LIN {X 0,Y 354.797,Z 576.907,A -85,B 0,C 180,E1 -13637.677,E2 -13637.677} C_VEL
LIN {X 0,Y 353.778,Z 635.743,A -85,B 0,C 180,E1 -13639.096,E2 -13639.096} C_VEL
LIN {X 0,Y 353.628,Z 649.216,A -85,B 0,C 180,E1 -13639.603,E2 -13639.603} C_VEL
LIN {X 0,Y 353.219,Z 662.716,A -85,B 0,C 180,E1 -13640.361,E2 -13640.361} C_VEL
LIN {X 0,Y 352.689,Z 674.449,A -85,B 0,C 180,E1 -13641.241,E2 -13641.241} C_VEL
LIN {X 0,Y 352.081,Z 686.1,A -85,B 0,C 180,E1 -13642.369,E2 -13642.369} C_VEL
LIN {X 0,Y 351.35,Z 696.823,A -85,B 0,C 180,E1 -13643.659,E2 -13643.659} C_VEL
LIN {X 0,Y 350.663,Z 705.588,A -85,B 0,C 180,E1 -13644.945,E2 -13644.945} C_VEL
LIN {X 0,Y 349.989,Z 714.199,A -85,B 0,C 180,E1 -13646.481,E2 -13646.481} C_VEL
LIN {X 0,Y 349.423,Z 721.312,A -85,B 0,C 180,E1 -13648.03,E2 -13648.03} C_VEL
LIN {X 0,Y 348.756,Z 728.774,A -85,B 0,C 180,E1 -13650.053,E2 -13650.053} C_VEL
LIN {X 0,Y 348.488,Z 733.524,A -85,B 0,C 180,E1 -13651.71,E2 -13651.71} C_VEL
LIN {X 0,Y 348.166,Z 737.758,A -85,B 0,C 180,E1 -13653.635,E2 -13653.635} C_VEL
LIN {X 0,Y 348.044,Z 740.417,A -85,B 0,C 180,E1 -13655.319,E2 -13655.319} C_VEL
LIN {X 0,Y 348.012,Z 742.443,A -85,B 0,C 180,E1 -13657.437,E2 -13657.437} C_VEL
LIN {X 0,Y 348.114,Z 743.004,A -85,B 0,C 180,E1 -13658.691,E2 -13658.691} C_VEL
LIN {X 0,Y 348.273,Z 743.074,A -85,B 0,C 180,E1 -13659.937,E2 -13659.937} C_VEL
LIN {X 0,Y 348.516,Z 742.538,A -85,B 0,C 180,E1 -13661.396,E2 -13661.396} C_VEL
LIN {X 0,Y 348.724,Z 741.797,A -85,B 0,C 180,E1 -13662.404,E2 -13662.404} C_VEL
LIN {X 0,Y 349.092,Z 740.415,A -85,B 0,C 180,E1 -13663.629,E2 -13663.629} C_VEL
LIN {X 0,Y 349.712,Z 737.457,A -85,B 0,C 180,E1 -13665.451,E2 -13665.451} C_VEL
LIN {X 0,Y 350.505,Z 733.331,A -85,B 0,C 180,E1 -13667.258,E2 -13667.258} C_VEL
LIN {X 0,Y 351.534,Z 727.601,A -85,B 0,C 180,E1 -13669.148,E2 -13669.148} C_VEL
LIN {X 0,Y 352.555,Z 721.084,A -85,B 0,C 180,E1 -13670.823,E2 -13670.823} C_VEL
LIN {X 0,Y 353.791,Z 712.466,A -85,B 0,C 180,E1 -13672.582,E2 -13672.582} C_VEL
LIN {X 0,Y 354.949,Z 703.421,A -85,B 0,C 180,E1 -13674.064,E2 -13674.064} C_VEL
LIN {X 0,Y 356.03,Z 693.807,A -85,B 0,C 180,E1 -13675.329,E2 -13675.329} C_VEL
LIN {X 0,Y 357.056,Z 682.997,A -85,B 0,C 180,E1 -13676.473,E2 -13676.473} C_VEL
LIN {X 0,Y 357.886,Z 671.118,A -85,B 0,C 180,E1 -13677.468,E2 -13677.468} C_VEL
LIN {X 0,Y 358.466,Z 657.986,A -85,B 0,C 180,E1 -13678.284,E2 -13678.284} C_VEL
LIN {X 0,Y 358.763,Z 645.264,A -85,B 0,C 180,E1 -13678.843,E2 -13678.843} C_VEL
LIN {X 0,Y 359.132,Z 620.722,A -85,B 0,C 180,E1 -13679.534,E2 -13679.534} C_VEL
LIN {X 0,Y 360.495,Z 582.186,A -85,B 0,C 180,E1 -13680.545,E2 -13680.545} C_VEL
LIN {X 0,Y 354.117,Z 568.659,A -85,B 0,C 180,E1 -13681.601,E2 -13681.601} C_VEL
LIN {X 0,Y 349.417,Z 560.316,A -85,B 0,C 180,E1 -13682.383,E2 -13682.383} C_VEL
LIN {X 0,Y 348.227,Z 557.698,A -85,B 0,C 180,E1 -13682.603,E2 -13682.603} C_VEL
LIN {X 0,Y 348.11,Z 557.127,A -85,B 0,C 180,E1 -13682.676,E2 -13682.676} C_VEL
LIN {X 0,Y 348.099,Z 557.121,A -85,B 0,C 180,E1 -13686.958,E2 -13686.958} C_VEL
LIN {X 0,Y 347.959,Z 557.14,A -85,B 0,C 180,E1 -13689.299,E2 -13689.299} C_VEL
LIN {X 0,Y 347.884,Z 557.146,A -85,B 0,C 180,E1 -13692.84,E2 -13692.84} C_VEL
LIN {X 0,Y 347.829,Z 557.152,A -85,B 0,C 180,E1 -13696.432,E2 -13696.432} C_VEL
LIN {X 0,Y 347.846,Z 557.158,A -85,B 0,C 180,E1 -13698.861,E2 -13698.861} C_VEL
LIN {X 0,Y 347.765,Z 557.166,A -85,B 0,C 180,E1 -13702.58,E2 -13702.58} C_VEL
LIN {X 0,Y 347.803,Z 557.162,A -85,B 0,C 180,E1 -13705.109,E2 -13705.109} C_VEL
LIN {X 0,Y 347.803,Z 557.158,A -85,B 0,C 180,E1 -13707.695,E2 -13707.695} C_VEL
LIN {X 0,Y 347.756,Z 557.168,A -85,B 0,C 180,E1 -13710.347,E2 -13710.347} C_VEL
LIN {X 0,Y 347.736,Z 557.164,A -85,B 0,C 180,E1 -13714.465,E2 -13714.465} C_VEL
LIN {X 0,Y 347.769,Z 557.161,A -85,B 0,C 180,E1 -13717.99,E2 -13717.99} C_VEL
LIN {X 0,Y 347.778,Z 557.167,A -85,B 0,C 180,E1 -13721.61,E2 -13721.61} C_VEL
LIN {X 0,Y 347.825,Z 557.158,A -85,B 0,C 180,E1 -13725.007,E2 -13725.007} C_VEL
LIN {X 0,Y 347.779,Z 557.165,A -85,B 0,C 180,E1 -13728.392,E2 -13728.392} C_VEL
LIN {X 0,Y 347.801,Z 557.245,A -85,B 0,C 180,E1 -13731.216,E2 -13731.216} C_VEL
LIN {X 0,Y 351.006,Z 568.194,A -85,B 0,C 180,E1 -13734.506,E2 -13734.506} C_VEL
LIN {X 0,Y 353.622,Z 578.805,A -85,B 0,C 180,E1 -13737.302,E2 -13737.302} C_VEL
LIN {X 0,Y 355.347,Z 587.427,A -85,B 0,C 180,E1 -13739.386,E2 -13739.386} C_VEL
LIN {X 0,Y 355.219,Z 590.506,A -85,B 0,C 180,E1 -13740.03,E2 -13740.03} C_VEL
LIN {X 0,Y 352.496,Z 610.75,A -85,B 0,C 180,E1 -13743.985,E2 -13743.985} C_VEL
LIN {X 0,Y 351.698,Z 617.716,A -85,B 0,C 180,E1 -13745.318,E2 -13745.318} C_VEL
LIN {X 0,Y 355.284,Z 641.232,A -85,B 0,C 180,E1 -13746.39,E2 -13746.39} C_VEL
LIN {X 0,Y 357.422,Z 662.797,A -85,B 0,C 180,E1 -13747.201,E2 -13747.201} C_VEL
LIN {X 0,Y 358.192,Z 678.894,A -85,B 0,C 180,E1 -13747.723,E2 -13747.723} C_VEL
LIN {X 0,Y 356.353,Z 732.757,A -85,B 0,C 180,E1 -13749.097,E2 -13749.097} C_VEL
LIN {X 0,Y 355.4,Z 746.792,A -85,B 0,C 180,E1 -13749.679,E2 -13749.679} C_VEL
LIN {X 0,Y 355.085,Z 750.828,A -85,B 0,C 180,E1 -13749.849,E2 -13749.849} C_VEL
LIN {X 0,Y 354.525,Z 764.15,A -85,B 0,C 180,E1 -13750.269,E2 -13750.269} C_VEL
LIN {X 0,Y 353.732,Z 776.246,A -85,B 0,C 180,E1 -13750.865,E2 -13750.865} C_VEL
LIN {X 0,Y 352.774,Z 788.474,A -85,B 0,C 180,E1 -13751.715,E2 -13751.715} C_VEL
LIN {X 0,Y 351.717,Z 799.465,A -85,B 0,C 180,E1 -13752.71,E2 -13752.71} C_VEL
LIN {X 0,Y 350.555,Z 810.407,A -85,B 0,C 180,E1 -13753.965,E2 -13753.965} C_VEL
LIN {X 0,Y 349.407,Z 820.549,A -85,B 0,C 180,E1 -13755.439,E2 -13755.439} C_VEL
LIN {X 0,Y 348.514,Z 828.654,A -85,B 0,C 180,E1 -13756.889,E2 -13756.889} C_VEL
LIN {X 0,Y 347.567,Z 836.584,A -85,B 0,C 180,E1 -13758.631,E2 -13758.631} C_VEL
LIN {X 0,Y 347.055,Z 841.938,A -85,B 0,C 180,E1 -13760.09,E2 -13760.09} C_VEL
LIN {X 0,Y 346.613,Z 847.165,A -85,B 0,C 180,E1 -13761.841,E2 -13761.841} C_VEL
LIN {X 0,Y 346.333,Z 851.786,A -85,B 0,C 180,E1 -13763.902,E2 -13763.902} C_VEL
LIN {X 0,Y 346.288,Z 854.185,A -85,B 0,C 180,E1 -13765.345,E2 -13765.345} C_VEL
LIN {X 0,Y 346.225,Z 855.612,A -85,B 0,C 180,E1 -13766.51,E2 -13766.51} C_VEL
LIN {X 0,Y 346.248,Z 857.236,A -85,B 0,C 180,E1 -13768.838,E2 -13768.838} C_VEL
LIN {X 0,Y 346.311,Z 857.456,A -85,B 0,C 180,E1 -13770.001,E2 -13770.001} C_VEL
LIN {X 0,Y 346.228,Z 857.23,A -85,B 0,C 180,E1 -13771.164,E2 -13771.164} C_VEL
LIN {X 0,Y 346.216,Z 855.598,A -85,B 0,C 180,E1 -13773.492,E2 -13773.492} C_VEL
LIN {X 0,Y 346.279,Z 854.163,A -85,B 0,C 180,E1 -13774.657,E2 -13774.657} C_VEL
LIN {X 0,Y 346.307,Z 851.838,A -85,B 0,C 180,E1 -13776.058,E2 -13776.058} C_VEL
LIN {X 0,Y 346.61,Z 847.128,A -85,B 0,C 180,E1 -13778.161,E2 -13778.161} C_VEL
LIN {X 0,Y 347.137,Z 840.879,A -85,B 0,C 180,E1 -13780.205,E2 -13780.205} C_VEL
LIN {X 0,Y 347.798,Z 834.061,A -85,B 0,C 180,E1 -13781.955,E2 -13781.955} C_VEL
LIN {X 0,Y 348.86,Z 825.532,A -85,B 0,C 180,E1 -13783.693,E2 -13783.693} C_VEL
LIN {X 0,Y 349.858,Z 816.746,A -85,B 0,C 180,E1 -13785.139,E2 -13785.139} C_VEL
LIN {X 0,Y 350.833,Z 807.081,A -85,B 0,C 180,E1 -13786.437,E2 -13786.437} C_VEL
LIN {X 0,Y 351.991,Z 796.48,A -85,B 0,C 180,E1 -13787.578,E2 -13787.578} C_VEL
LIN {X 0,Y 353.108,Z 784.571,A -85,B 0,C 180,E1 -13788.57,E2 -13788.57} C_VEL
LIN {X 0,Y 353.992,Z 772.163,A -85,B 0,C 180,E1 -13789.349,E2 -13789.349} C_VEL
LIN {X 0,Y 354.749,Z 760.169,A -85,B 0,C 180,E1 -13789.871,E2 -13789.871} C_VEL
LIN {X 0,Y 355.231,Z 746.868,A -85,B 0,C 180,E1 -13790.22,E2 -13790.22} C_VEL
LIN {X 0,Y 356.311,Z 677.092,A -85,B 0,C 180,E1 -13791.622,E2 -13791.622} C_VEL
LIN {X 0,Y 352.473,Z 643.046,A -85,B 0,C 180,E1 -13792.599,E2 -13792.599} C_VEL
LIN {X 0,Y 351.528,Z 636.097,A -85,B 0,C 180,E1 -13792.83,E2 -13792.83} C_VEL
LIN {X 0,Y 350.218,Z 619.795,A -85,B 0,C 180,E1 -13793.899,E2 -13793.899} C_VEL
LIN {X 0,Y 352.061,Z 599.692,A -85,B 0,C 180,E1 -13797.978,E2 -13797.978} C_VEL
LIN {X 0,Y 353.609,Z 584.378,A -85,B 0,C 180,E1 -13801.115,E2 -13801.115} C_VEL
LIN {X 0,Y 351.574,Z 574.031,A -85,B 0,C 180,E1 -13803.456,E2 -13803.456} C_VEL
LIN {X 0,Y 348.306,Z 559.575,A -85,B 0,C 180,E1 -13806.864,E2 -13806.864} C_VEL
LIN {X 0,Y 347.787,Z 557.165,A -85,B 0,C 180,E1 -13807.485,E2 -13807.485} C_VEL
LIN {X 0,Y 347.735,Z 557.17,A -85,B 0,C 180,E1 -13810.297,E2 -13810.297} C_VEL
LIN {X 0,Y 347.725,Z 557.162,A -85,B 0,C 180,E1 -13813.408,E2 -13813.408} C_VEL
LIN {X 0,Y 347.73,Z 557.171,A -85,B 0,C 180,E1 -13816.686,E2 -13816.686} C_VEL
LIN {X 0,Y 347.749,Z 557.166,A -85,B 0,C 180,E1 -13820.173,E2 -13820.173} C_VEL
LIN {X 0,Y 347.764,Z 557.157,A -85,B 0,C 180,E1 -13822.679,E2 -13822.679} C_VEL
LIN {X 0,Y 347.75,Z 557.167,A -85,B 0,C 180,E1 -13825.956,E2 -13825.956} C_VEL
LIN {X 0,Y 347.765,Z 557.153,A -85,B 0,C 180,E1 -13829.654,E2 -13829.654} C_VEL
LIN {X 0,Y 347.853,Z 557.154,A -85,B 0,C 180,E1 -13832.745,E2 -13832.745} C_VEL
LIN {X 0,Y 347.787,Z 557.151,A -85,B 0,C 180,E1 -13836.162,E2 -13836.162} C_VEL
LIN {X 0,Y 347.808,Z 557.155,A -85,B 0,C 180,E1 -13839.909,E2 -13839.909} C_VEL
LIN {X 0,Y 347.867,Z 557.131,A -85,B 0,C 180,E1 -13842.359,E2 -13842.359} C_VEL
LIN {X 0,Y 347.899,Z 557.148,A -85,B 0,C 180,E1 -13845.971,E2 -13845.971} C_VEL
LIN {X 0,Y 347.929,Z 557.124,A -85,B 0,C 180,E1 -13849.526,E2 -13849.526} C_VEL
LIN {X 0,Y 348.093,Z 557.123,A -85,B 0,C 180,E1 -13853.042,E2 -13853.042} C_VEL
LIN {X 0,Y 348.206,Z 557.089,A -85,B 0,C 180,E1 -13857.687,E2 -13857.687} C_VEL
LIN {X 0,Y 348.325,Z 557.095,A -85,B 0,C 180,E1 -13860,E2 -13860} C_VEL
LIN {X 0,Y 348.207,Z 557.106,A -85,B 0,C 180,E1 -13862.314,E2 -13862.314} C_VEL
LIN {X 0,Y 348.094,Z 557.116,A -85,B 0,C 180,E1 -13866.958,E2 -13866.958} C_VEL
LIN {X 0,Y 347.931,Z 557.137,A -85,B 0,C 180,E1 -13870.474,E2 -13870.474} C_VEL
LIN {X 0,Y 347.9,Z 557.141,A -85,B 0,C 180,E1 -13874.15,E2 -13874.15} C_VEL
LIN {X 0,Y 347.892,Z 557.135,A -85,B 0,C 180,E1 -13878.29,E2 -13878.29} C_VEL
LIN {X 0,Y 347.79,Z 557.16,A -85,B 0,C 180,E1 -13881.635,E2 -13881.635} C_VEL
LIN {X 0,Y 347.813,Z 557.145,A -85,B 0,C 180,E1 -13885.108,E2 -13885.108} C_VEL
LIN {X 0,Y 347.81,Z 557.159,A -85,B 0,C 180,E1 -13887.694,E2 -13887.694} C_VEL
LIN {X 0,Y 347.751,Z 557.156,A -85,B 0,C 180,E1 -13890.348,E2 -13890.348} C_VEL
LIN {X 0,Y 347.75,Z 557.168,A -85,B 0,C 180,E1 -13894.044,E2 -13894.044} C_VEL
LIN {X 0,Y 347.763,Z 557.167,A -85,B 0,C 180,E1 -13897.321,E2 -13897.321} C_VEL
LIN {X 0,Y 347.734,Z 557.167,A -85,B 0,C 180,E1 -13900.297,E2 -13900.297} C_VEL
LIN {X 0,Y 347.725,Z 557.163,A -85,B 0,C 180,E1 -13903.408,E2 -13903.408} C_VEL
LIN {X 0,Y 347.727,Z 557.152,A -85,B 0,C 180,E1 -13906.686,E2 -13906.686} C_VEL
LIN {X 0,Y 347.751,Z 557.17,A -85,B 0,C 180,E1 -13910.173,E2 -13910.173} C_VEL
LIN {X 0,Y 347.765,Z 557.155,A -85,B 0,C 180,E1 -13912.679,E2 -13912.679} C_VEL
LIN {X 0,Y 347.804,Z 557.278,A -85,B 0,C 180,E1 -13915.058,E2 -13915.058} C_VEL
LIN {X 0,Y 351.695,Z 571.483,A -85,B 0,C 180,E1 -13918.025,E2 -13918.025} C_VEL
LIN {X 0,Y 354.731,Z 584.606,A -85,B 0,C 180,E1 -13920.662,E2 -13920.662} C_VEL
LIN {X 0,Y 355.49,Z 588.601,A -85,B 0,C 180,E1 -13921.437,E2 -13921.437} C_VEL
LIN {X 0,Y 354.195,Z 606.433,A -85,B 0,C 180,E1 -13924.432,E2 -13924.432} C_VEL
LIN {X 0,Y 353.21,Z 623.88,A -85,B 0,C 180,E1 -13927.211,E2 -13927.211} C_VEL
LIN {X 0,Y 357.261,Z 649.9,A -85,B 0,C 180,E1 -13928.051,E2 -13928.051} C_VEL
LIN {X 0,Y 355.98,Z 721.054,A -85,B 0,C 180,E1 -13929.486,E2 -13929.486} C_VEL
LIN {X 0,Y 355.648,Z 737.977,A -85,B 0,C 180,E1 -13929.881,E2 -13929.881} C_VEL
LIN {X 0,Y 354.963,Z 751.645,A -85,B 0,C 180,E1 -13930.443,E2 -13930.443} C_VEL
LIN {X 0,Y 354.078,Z 763.979,A -85,B 0,C 180,E1 -13931.183,E2 -13931.183} C_VEL
LIN {X 0,Y 353.008,Z 776.117,A -85,B 0,C 180,E1 -13932.175,E2 -13932.175} C_VEL
LIN {X 0,Y 351.907,Z 787.509,A -85,B 0,C 180,E1 -13933.377,E2 -13933.377} C_VEL
LIN {X 0,Y 350.973,Z 796.862,A -85,B 0,C 180,E1 -13934.615,E2 -13934.615} C_VEL
LIN {X 0,Y 349.814,Z 805.738,A -85,B 0,C 180,E1 -13936.048,E2 -13936.048} C_VEL
LIN {X 0,Y 348.749,Z 814.393,A -85,B 0,C 180,E1 -13937.783,E2 -13937.783} C_VEL
LIN {X 0,Y 347.875,Z 821.352,A -85,B 0,C 180,E1 -13939.523,E2 -13939.523} C_VEL
LIN {X 0,Y 347.175,Z 826.884,A -85,B 0,C 180,E1 -13941.266,E2 -13941.266} C_VEL
LIN {X 0,Y 346.719,Z 831.878,A -85,B 0,C 180,E1 -13943.333,E2 -13943.333} C_VEL
LIN {X 0,Y 346.422,Z 835.356,A -85,B 0,C 180,E1 -13945.344,E2 -13945.344} C_VEL
LIN {X 0,Y 346.254,Z 836.779,A -85,B 0,C 180,E1 -13946.508,E2 -13946.508} C_VEL
LIN {X 0,Y 346.155,Z 838.388,A -85,B 0,C 180,E1 -13948.836,E2 -13948.836} C_VEL
LIN {X 0,Y 346.167,Z 838.622,A -85,B 0,C 180,E1 -13949.999,E2 -13949.999} C_VEL
LIN {X 0,Y 346.155,Z 838.431,A -85,B 0,C 180,E1 -13951.162,E2 -13951.162} C_VEL
LIN {X 0,Y 346.246,Z 836.878,A -85,B 0,C 180,E1 -13953.49,E2 -13953.49} C_VEL
LIN {X 0,Y 346.419,Z 835.511,A -85,B 0,C 180,E1 -13954.654,E2 -13954.654} C_VEL
LIN {X 0,Y 346.714,Z 832.104,A -85,B 0,C 180,E1 -13956.661,E2 -13956.661} C_VEL
LIN {X 0,Y 347.167,Z 827.164,A -85,B 0,C 180,E1 -13958.732,E2 -13958.732} C_VEL
LIN {X 0,Y 347.836,Z 821.709,A -85,B 0,C 180,E1 -13960.476,E2 -13960.476} C_VEL
LIN {X 0,Y 348.677,Z 814.868,A -85,B 0,C 180,E1 -13962.217,E2 -13962.217} C_VEL
LIN {X 0,Y 349.756,Z 806.294,A -85,B 0,C 180,E1 -13963.952,E2 -13963.952} C_VEL
LIN {X 0,Y 350.883,Z 797.67,A -85,B 0,C 180,E1 -13965.364,E2 -13965.364} C_VEL
LIN {X 0,Y 351.847,Z 788.574,A -85,B 0,C 180,E1 -13966.594,E2 -13966.594} C_VEL
LIN {X 0,Y 352.816,Z 778.694,A -85,B 0,C 180,E1 -13967.683,E2 -13967.683} C_VEL
LIN {X 0,Y 353.861,Z 767.21,A -85,B 0,C 180,E1 -13968.677,E2 -13968.677} C_VEL
LIN {X 0,Y 354.864,Z 754.229,A -85,B 0,C 180,E1 -13969.523,E2 -13969.523} C_VEL
LIN {X 0,Y 355.476,Z 741.857,A -85,B 0,C 180,E1 -13970.09,E2 -13970.09} C_VEL
LIN {X 0,Y 355.91,Z 727.81,A -85,B 0,C 180,E1 -13970.479,E2 -13970.479} C_VEL
LIN {X 0,Y 356.196,Z 714.351,A -85,B 0,C 180,E1 -13970.747,E2 -13970.747} C_VEL
LIN {X 0,Y 355.83,Z 708.537,A -85,B 0,C 180,E1 -13970.893,E2 -13970.893} C_VEL
LIN {X 0,Y 353.319,Z 699.198,A -85,B 0,C 180,E1 -13971.25,E2 -13971.25} C_VEL
LIN {X 0,Y 350.713,Z 689.862,A -85,B 0,C 180,E1 -13971.618,E2 -13971.618} C_VEL
LIN {X 0,Y 350.198,Z 684.045,A -85,B 0,C 180,E1 -13971.778,E2 -13971.778} C_VEL
LIN {X 0,Y 350.61,Z 652.041,A -85,B 0,C 180,E1 -13972.448,E2 -13972.448} C_VEL
LIN {X 0,Y 346.314,Z 627.329,A -85,B 0,C 180,E1 -13973.291,E2 -13973.291} C_VEL
LIN {X 0,Y 345.82,Z 624.898,A -85,B 0,C 180,E1 -13973.381,E2 -13973.381} C_VEL
LIN {X 0,Y 347.067,Z 605.912,A -85,B 0,C 180,E1 -13976.806,E2 -13976.806} C_VEL
LIN {X 0,Y 348.183,Z 590.44,A -85,B 0,C 180,E1 -13979.779,E2 -13979.779} C_VEL
LIN {X 0,Y 347.335,Z 584.737,A -85,B 0,C 180,E1 -13981.015,E2 -13981.015} C_VEL
LIN {X 0,Y 344.655,Z 572.639,A -85,B 0,C 180,E1 -13983.754,E2 -13983.754} C_VEL
LIN {X 0,Y 341.343,Z 560.29,A -85,B 0,C 180,E1 -13986.66,E2 -13986.66} C_VEL
LIN {X 0,Y 340.74,Z 558.045,A -85,B 0,C 180,E1 -13987.197,E2 -13987.197} C_VEL
LIN {X 0,Y 340.682,Z 558.052,A -85,B 0,C 180,E1 -13991.308,E2 -13991.308} C_VEL
LIN {X 0,Y 340.739,Z 558.039,A -85,B 0,C 180,E1 -13995.47,E2 -13995.47} C_VEL
LIN {X 0,Y 340.769,Z 558.037,A -85,B 0,C 180,E1 -13996.475,E2 -13996.475} C_VEL
LIN {X 0,Y 348.026,Z 579.157,A -85,B 0,C 180,E1 -13997.408,E2 -13997.408} C_VEL
LIN {X 0,Y 346.904,Z 634.659,A -85,B 0,C 180,E1 -13998.769,E2 -13998.769} C_VEL
LIN {X 0,Y 346.806,Z 648.393,A -85,B 0,C 180,E1 -13999.264,E2 -13999.264} C_VEL
LIN {X 0,Y 346.437,Z 661.709,A -85,B 0,C 180,E1 -13999.991,E2 -13999.991} C_VEL
LIN {X 0,Y 345.809,Z 674.596,A -85,B 0,C 180,E1 -14000.948,E2 -14000.948} C_VEL
LIN {X 0,Y 345.225,Z 685.475,A -85,B 0,C 180,E1 -14001.988,E2 -14001.988} C_VEL
LIN {X 0,Y 344.473,Z 696.947,A -85,B 0,C 180,E1 -14003.368,E2 -14003.368} C_VEL
LIN {X 0,Y 343.661,Z 707.135,A -85,B 0,C 180,E1 -14004.884,E2 -14004.884} C_VEL
LIN {X 0,Y 342.855,Z 716.569,A -85,B 0,C 180,E1 -14006.642,E2 -14006.642} C_VEL
LIN {X 0,Y 342.239,Z 724.267,A -85,B 0,C 180,E1 -14008.422,E2 -14008.422} C_VEL
LIN {X 0,Y 341.643,Z 731.044,A -85,B 0,C 180,E1 -14010.415,E2 -14010.415} C_VEL
LIN {X 0,Y 341.374,Z 735.933,A -85,B 0,C 180,E1 -14012.279,E2 -14012.279} C_VEL
LIN {X 0,Y 341.046,Z 739.996,A -85,B 0,C 180,E1 -14014.358,E2 -14014.358} C_VEL
LIN {X 0,Y 340.994,Z 741.786,A -85,B 0,C 180,E1 -14015.656,E2 -14015.656} C_VEL
LIN {X 0,Y 340.988,Z 743.081,A -85,B 0,C 180,E1 -14016.946,E2 -14016.946} C_VEL
LIN {X 0,Y 341.043,Z 743.879,A -85,B 0,C 180,E1 -14018.227,E2 -14018.227} C_VEL
LIN {X 0,Y 341.185,Z 744.159,A -85,B 0,C 180,E1 -14019.502,E2 -14019.502} C_VEL
LIN {X 0,Y 341.466,Z 743.8,A -85,B 0,C 180,E1 -14021.215,E2 -14021.215} C_VEL
LIN {X 0,Y 342.005,Z 742.182,A -85,B 0,C 180,E1 -14023.28,E2 -14023.28} C_VEL
LIN {X 0,Y 342.459,Z 740.319,A -85,B 0,C 180,E1 -14024.689,E2 -14024.689} C_VEL
LIN {X 0,Y 343.13,Z 737.212,A -85,B 0,C 180,E1 -14026.376,E2 -14026.376} C_VEL
LIN {X 0,Y 344.212,Z 731.735,A -85,B 0,C 180,E1 -14028.526,E2 -14028.526} C_VEL
LIN {X 0,Y 345.34,Z 725.653,A -85,B 0,C 180,E1 -14030.334,E2 -14030.334} C_VEL
LIN {X 0,Y 346.572,Z 717.914,A -85,B 0,C 180,E1 -14032.133,E2 -14032.133} C_VEL
LIN {X 0,Y 347.775,Z 709.63,A -85,B 0,C 180,E1 -14033.677,E2 -14033.677} C_VEL
LIN {X 0,Y 348.945,Z 700.308,A -85,B 0,C 180,E1 -14035.09,E2 -14035.09} C_VEL
LIN {X 0,Y 350.17,Z 689.347,A -85,B 0,C 180,E1 -14036.404,E2 -14036.404} C_VEL
LIN {X 0,Y 351.207,Z 677.219,A -85,B 0,C 180,E1 -14037.563,E2 -14037.563} C_VEL
LIN {X 0,Y 352.016,Z 664.559,A -85,B 0,C 180,E1 -14038.47,E2 -14038.47} C_VEL
LIN {X 0,Y 352.454,Z 651.997,A -85,B 0,C 180,E1 -14039.137,E2 -14039.137} C_VEL
LIN {X 0,Y 352.605,Z 637.701,A -85,B 0,C 180,E1 -14039.632,E2 -14039.632} C_VEL
LIN {X 0,Y 353.678,Z 601.91,A -85,B 0,C 180,E1 -14040.603,E2 -14040.603} C_VEL
LIN {X 0,Y 354.281,Z 584.167,A -85,B 0,C 180,E1 -14041.092,E2 -14041.092} C_VEL
LIN {X 0,Y 348.798,Z 572.457,A -85,B 0,C 180,E1 -14042.053,E2 -14042.053} C_VEL
LIN {X 0,Y 342.873,Z 562.026,A -85,B 0,C 180,E1 -14043.085,E2 -14043.085} C_VEL
LIN {X 0,Y 341.244,Z 559.432,A -85,B 0,C 180,E1 -14043.376,E2 -14043.376} C_VEL
LIN {X 0,Y 340.924,Z 558.018,A -85,B 0,C 180,E1 -14043.472,E2 -14043.472} C_VEL
LIN {X 0,Y 341.068,Z 557.996,A -85,B 0,C 180,E1 -14047.102,E2 -14047.102} C_VEL
LIN {X 0,Y 340.865,Z 558.022,A -85,B 0,C 180,E1 -14050.694,E2 -14050.694} C_VEL
LIN {X 0,Y 340.853,Z 558.028,A -85,B 0,C 180,E1 -14054.325,E2 -14054.325} C_VEL
LIN {X 0,Y 340.828,Z 558.03,A -85,B 0,C 180,E1 -14058.467,E2 -14058.467} C_VEL
LIN {X 0,Y 340.744,Z 558.04,A -85,B 0,C 180,E1 -14061.858,E2 -14061.858} C_VEL
LIN {X 0,Y 340.764,Z 558.036,A -85,B 0,C 180,E1 -14065.665,E2 -14065.665} C_VEL
LIN {X 0,Y 340.733,Z 558.041,A -85,B 0,C 180,E1 -14068.32,E2 -14068.32} C_VEL
LIN {X 0,Y 340.696,Z 558.047,A -85,B 0,C 180,E1 -14071.045,E2 -14071.045} C_VEL
LIN {X 0,Y 340.711,Z 558.041,A -85,B 0,C 180,E1 -14075.28,E2 -14075.28} C_VEL
LIN {X 0,Y 340.711,Z 558.043,A -85,B 0,C 180,E1 -14078.389,E2 -14078.389} C_VEL
LIN {X 0,Y 340.719,Z 558.047,A -85,B 0,C 180,E1 -14081.305,E2 -14081.305} C_VEL
LIN {X 0,Y 340.776,Z 558.037,A -85,B 0,C 180,E1 -14084.524,E2 -14084.524} C_VEL
LIN {X 0,Y 340.746,Z 558.042,A -85,B 0,C 180,E1 -14087.946,E2 -14087.946} C_VEL
LIN {X 0,Y 340.772,Z 558.177,A -85,B 0,C 180,E1 -14090.349,E2 -14090.349} C_VEL
LIN {X 0,Y 343.461,Z 567.325,A -85,B 0,C 180,E1 -14093.284,E2 -14093.284} C_VEL
LIN {X 0,Y 345.983,Z 576.696,A -85,B 0,C 180,E1 -14095.959,E2 -14095.959} C_VEL
LIN {X 0,Y 348.246,Z 587.4,A -85,B 0,C 180,E1 -14098.692,E2 -14098.692} C_VEL
LIN {X 0,Y 348.7,Z 590.418,A -85,B 0,C 180,E1 -14099.41,E2 -14099.41} C_VEL
LIN {X 0,Y 345.888,Z 610.163,A -85,B 0,C 180,E1 -14103.384,E2 -14103.384} C_VEL
LIN {X 0,Y 345.119,Z 616.67,A -85,B 0,C 180,E1 -14104.623,E2 -14104.623} C_VEL
LIN {X 0,Y 348.549,Z 638.007,A -85,B 0,C 180,E1 -14105.648,E2 -14105.648} C_VEL
LIN {X 0,Y 350.735,Z 658.092,A -85,B 0,C 180,E1 -14106.469,E2 -14106.469} C_VEL
LIN {X 0,Y 351.924,Z 678.447,A -85,B 0,C 180,E1 -14107.186,E2 -14107.186} C_VEL
LIN {X 0,Y 349.967,Z 731.889,A -85,B 0,C 180,E1 -14108.579,E2 -14108.579} C_VEL
LIN {X 0,Y 349,Z 745.12,A -85,B 0,C 180,E1 -14109.135,E2 -14109.135} C_VEL
LIN {X 0,Y 348.391,Z 752.187,A -85,B 0,C 180,E1 -14109.483,E2 -14109.483} C_VEL
LIN {X 0,Y 347.823,Z 764.91,A -85,B 0,C 180,E1 -14109.911,E2 -14109.911} C_VEL
LIN {X 0,Y 346.952,Z 777.23,A -85,B 0,C 180,E1 -14110.553,E2 -14110.553} C_VEL
LIN {X 0,Y 345.872,Z 790.055,A -85,B 0,C 180,E1 -14111.49,E2 -14111.49} C_VEL
LIN {X 0,Y 344.806,Z 800.703,A -85,B 0,C 180,E1 -14112.505,E2 -14112.505} C_VEL
LIN {X 0,Y 343.665,Z 810.633,A -85,B 0,C 180,E1 -14113.692,E2 -14113.692} C_VEL
LIN {X 0,Y 342.527,Z 820.364,A -85,B 0,C 180,E1 -14115.14,E2 -14115.14} C_VEL
LIN {X 0,Y 341.578,Z 828.467,A -85,B 0,C 180,E1 -14116.618,E2 -14116.618} C_VEL
LIN {X 0,Y 340.569,Z 836.395,A -85,B 0,C 180,E1 -14118.394,E2 -14118.394} C_VEL
LIN {X 0,Y 340.038,Z 841.748,A -85,B 0,C 180,E1 -14119.883,E2 -14119.883} C_VEL
LIN {X 0,Y 339.564,Z 846.974,A -85,B 0,C 180,E1 -14121.671,E2 -14121.671} C_VEL
LIN {X 0,Y 339.252,Z 851.859,A -85,B 0,C 180,E1 -14123.922,E2 -14123.922} C_VEL
LIN {X 0,Y 339.185,Z 853.992,A -85,B 0,C 180,E1 -14125.247,E2 -14125.247} C_VEL
LIN {X 0,Y 339.149,Z 855.42,A -85,B 0,C 180,E1 -14126.437,E2 -14126.437} C_VEL
LIN {X 0,Y 339.147,Z 857.043,A -85,B 0,C 180,E1 -14128.814,E2 -14128.814} C_VEL
LIN {X 0,Y 339.213,Z 857.263,A -85,B 0,C 180,E1 -14130.001,E2 -14130.001} C_VEL
LIN {X 0,Y 339.127,Z 857.037,A -85,B 0,C 180,E1 -14131.188,E2 -14131.188} C_VEL
LIN {X 0,Y 339.14,Z 855.405,A -85,B 0,C 180,E1 -14133.565,E2 -14133.565} C_VEL
LIN {X 0,Y 339.174,Z 853.969,A -85,B 0,C 180,E1 -14134.755,E2 -14134.755} C_VEL
LIN {X 0,Y 339.262,Z 850.985,A -85,B 0,C 180,E1 -14136.543,E2 -14136.543} C_VEL
LIN {X 0,Y 339.558,Z 846.935,A -85,B 0,C 180,E1 -14138.331,E2 -14138.331} C_VEL
LIN {X 0,Y 340.113,Z 840.685,A -85,B 0,C 180,E1 -14140.418,E2 -14140.418} C_VEL
LIN {X 0,Y 340.821,Z 833.869,A -85,B 0,C 180,E1 -14142.203,E2 -14142.203} C_VEL
LIN {X 0,Y 341.935,Z 825.341,A -85,B 0,C 180,E1 -14143.976,E2 -14143.976} C_VEL
LIN {X 0,Y 342.968,Z 816.557,A -85,B 0,C 180,E1 -14145.45,E2 -14145.45} C_VEL
LIN {X 0,Y 343.995,Z 806.895,A -85,B 0,C 180,E1 -14146.774,E2 -14146.774} C_VEL
LIN {X 0,Y 345.207,Z 796.298,A -85,B 0,C 180,E1 -14147.935,E2 -14147.935} C_VEL
LIN {X 0,Y 346.377,Z 784.396,A -85,B 0,C 180,E1 -14148.945,E2 -14148.945} C_VEL
LIN {X 0,Y 347.305,Z 771.997,A -85,B 0,C 180,E1 -14149.737,E2 -14149.737} C_VEL
LIN {X 0,Y 348.098,Z 760.024,A -85,B 0,C 180,E1 -14150.267,E2 -14150.267} C_VEL
LIN {X 0,Y 348.597,Z 746.769,A -85,B 0,C 180,E1 -14150.622,E2 -14150.622} C_VEL
LIN {X 0,Y 349.646,Z 677.351,A -85,B 0,C 180,E1 -14152.048,E2 -14152.048} C_VEL
LIN {X 0,Y 345.99,Z 644.415,A -85,B 0,C 180,E1 -14153.014,E2 -14153.014} C_VEL
LIN {X 0,Y 344.786,Z 635.515,A -85,B 0,C 180,E1 -14153.329,E2 -14153.329} C_VEL
LIN {X 0,Y 343.393,Z 617.803,A -85,B 0,C 180,E1 -14154.525,E2 -14154.525} C_VEL
LIN {X 0,Y 345.254,Z 598.45,A -85,B 0,C 180,E1 -14158.541,E2 -14158.541} C_VEL
LIN {X 0,Y 346.622,Z 586.079,A -85,B 0,C 180,E1 -14161.132,E2 -14161.132} C_VEL
LIN {X 0,Y 345.282,Z 578.44,A -85,B 0,C 180,E1 -14162.876,E2 -14162.876} C_VEL
LIN {X 0,Y 342.197,Z 564.509,A -85,B 0,C 180,E1 -14166.19,E2 -14166.19} C_VEL
LIN {X 0,Y 340.737,Z 558.042,A -85,B 0,C 180,E1 -14167.805,E2 -14167.805} C_VEL
LIN {X 0,Y 340.688,Z 558.049,A -85,B 0,C 180,E1 -14171.31,E2 -14171.31} C_VEL
LIN {X 0,Y 340.684,Z 558.037,A -85,B 0,C 180,E1 -14174.539,E2 -14174.539} C_VEL
LIN {X 0,Y 340.701,Z 558.035,A -85,B 0,C 180,E1 -14177.955,E2 -14177.955} C_VEL
LIN {X 0,Y 340.735,Z 558.037,A -85,B 0,C 180,E1 -14181.773,E2 -14181.773} C_VEL
LIN {X 0,Y 340.725,Z 558.044,A -85,B 0,C 180,E1 -14185.596,E2 -14185.596} C_VEL
LIN {X 0,Y 340.705,Z 558.029,A -85,B 0,C 180,E1 -14188.956,E2 -14188.956} C_VEL
LIN {X 0,Y 340.78,Z 558.034,A -85,B 0,C 180,E1 -14192.474,E2 -14192.474} C_VEL
LIN {X 0,Y 340.756,Z 558.022,A -85,B 0,C 180,E1 -14195.638,E2 -14195.638} C_VEL
LIN {X 0,Y 340.736,Z 558.04,A -85,B 0,C 180,E1 -14199.473,E2 -14199.473} C_VEL
LIN {X 0,Y 340.859,Z 558.003,A -85,B 0,C 180,E1 -14201.984,E2 -14201.984} C_VEL
LIN {X 0,Y 340.871,Z 558.026,A -85,B 0,C 180,E1 -14205.705,E2 -14205.705} C_VEL
LIN {X 0,Y 340.872,Z 558.003,A -85,B 0,C 180,E1 -14209.306,E2 -14209.306} C_VEL
LIN {X 0,Y 341.061,Z 557.998,A -85,B 0,C 180,E1 -14212.898,E2 -14212.898} C_VEL
LIN {X 0,Y 341.168,Z 557.965,A -85,B 0,C 180,E1 -14217.639,E2 -14217.639} C_VEL
LIN {X 0,Y 341.276,Z 557.973,A -85,B 0,C 180,E1 -14220,E2 -14220} C_VEL
LIN {X 0,Y 341.169,Z 557.983,A -85,B 0,C 180,E1 -14222.361,E2 -14222.361} C_VEL
LIN {X 0,Y 341.062,Z 557.992,A -85,B 0,C 180,E1 -14227.102,E2 -14227.102} C_VEL
LIN {X 0,Y 340.873,Z 558.015,A -85,B 0,C 180,E1 -14230.694,E2 -14230.694} C_VEL
LIN {X 0,Y 340.864,Z 558.02,A -85,B 0,C 180,E1 -14234.325,E2 -14234.325} C_VEL
LIN {X 0,Y 340.838,Z 558.012,A -85,B 0,C 180,E1 -14238.466,E2 -14238.466} C_VEL
LIN {X 0,Y 340.755,Z 558.038,A -85,B 0,C 180,E1 -14241.857,E2 -14241.857} C_VEL
LIN {X 0,Y 340.774,Z 558.021,A -85,B 0,C 180,E1 -14245.664,E2 -14245.664} C_VEL
LIN {X 0,Y 340.73,Z 558.043,A -85,B 0,C 180,E1 -14248.321,E2 -14248.321} C_VEL
LIN {X 0,Y 340.7,Z 558.034,A -85,B 0,C 180,E1 -14251.045,E2 -14251.045} C_VEL
LIN {X 0,Y 340.72,Z 558.035,A -85,B 0,C 180,E1 -14255.279,E2 -14255.279} C_VEL
LIN {X 0,Y 340.712,Z 558.045,A -85,B 0,C 180,E1 -14258.386,E2 -14258.386} C_VEL
LIN {X 0,Y 340.701,Z 558.047,A -85,B 0,C 180,E1 -14262.045,E2 -14262.045} C_VEL
LIN {X 0,Y 340.654,Z 558.037,A -85,B 0,C 180,E1 -14266.227,E2 -14266.227} C_VEL
LIN {X 0,Y 340.691,Z 558.049,A -85,B 0,C 180,E1 -14269.753,E2 -14269.753} C_VEL
LIN {X 0,Y 340.708,Z 558.041,A -85,B 0,C 180,E1 -14273.258,E2 -14273.258} C_VEL
LIN {X 0,Y 340.767,Z 558.212,A -85,B 0,C 180,E1 -14274.5,E2 -14274.5} C_VEL
LIN {X 0,Y 344.653,Z 572.069,A -85,B 0,C 180,E1 -14277.467,E2 -14277.467} C_VEL
LIN {X 0,Y 347.902,Z 585.927,A -85,B 0,C 180,E1 -14280.302,E2 -14280.302} C_VEL
LIN {X 0,Y 348.788,Z 591.609,A -85,B 0,C 180,E1 -14281.408,E2 -14281.408} C_VEL
LIN {X 0,Y 347.161,Z 612.087,A -85,B 0,C 180,E1 -14284.841,E2 -14284.841} C_VEL
LIN {X 0,Y 346.504,Z 623.989,A -85,B 0,C 180,E1 -14286.746,E2 -14286.746} C_VEL
LIN {X 0,Y 350.693,Z 649.998,A -85,B 0,C 180,E1 -14287.618,E2 -14287.618} C_VEL
LIN {X 0,Y 349.362,Z 721.155,A -85,B 0,C 180,E1 -14289.079,E2 -14289.079} C_VEL
LIN {X 0,Y 349.002,Z 738.12,A -85,B 0,C 180,E1 -14289.48,E2 -14289.48} C_VEL
LIN {X 0,Y 348.289,Z 751.809,A -85,B 0,C 180,E1 -14290.053,E2 -14290.053} C_VEL
LIN {X 0,Y 347.364,Z 764.155,A -85,B 0,C 180,E1 -14290.805,E2 -14290.805} C_VEL
LIN {X 0,Y 346.273,Z 776.298,A -85,B 0,C 180,E1 -14291.816,E2 -14291.816} C_VEL
LIN {X 0,Y 345.113,Z 787.556,A -85,B 0,C 180,E1 -14293.023,E2 -14293.023} C_VEL
LIN {X 0,Y 344.124,Z 797.191,A -85,B 0,C 180,E1 -14294.323,E2 -14294.323} C_VEL
LIN {X 0,Y 342.936,Z 805.928,A -85,B 0,C 180,E1 -14295.763,E2 -14295.763} C_VEL
LIN {X 0,Y 341.806,Z 814.585,A -85,B 0,C 180,E1 -14297.531,E2 -14297.531} C_VEL
LIN {X 0,Y 340.875,Z 821.544,A -85,B 0,C 180,E1 -14299.306,E2 -14299.306} C_VEL
LIN {X 0,Y 340.14,Z 827.077,A -85,B 0,C 180,E1 -14301.084,E2 -14301.084} C_VEL
LIN {X 0,Y 339.729,Z 831.41,A -85,B 0,C 180,E1 -14302.869,E2 -14302.869} C_VEL
LIN {X 0,Y 339.497,Z 833.69,A -85,B 0,C 180,E1 -14304.058,E2 -14304.058} C_VEL
LIN {X 0,Y 339.342,Z 835.55,A -85,B 0,C 180,E1 -14305.247,E2 -14305.247} C_VEL
LIN {X 0,Y 339.182,Z 836.972,A -85,B 0,C 180,E1 -14306.435,E2 -14306.435} C_VEL
LIN {X 0,Y 339.058,Z 838.582,A -85,B 0,C 180,E1 -14308.811,E2 -14308.811} C_VEL
LIN {X 0,Y 339.07,Z 838.815,A -85,B 0,C 180,E1 -14309.999,E2 -14309.999} C_VEL
LIN {X 0,Y 339.057,Z 838.623,A -85,B 0,C 180,E1 -14311.187,E2 -14311.187} C_VEL
LIN {X 0,Y 339.175,Z 837.07,A -85,B 0,C 180,E1 -14313.563,E2 -14313.563} C_VEL
LIN {X 0,Y 339.339,Z 835.703,A -85,B 0,C 180,E1 -14314.751,E2 -14314.751} C_VEL
LIN {X 0,Y 339.612,Z 832.656,A -85,B 0,C 180,E1 -14316.623,E2 -14316.623} C_VEL
LIN {X 0,Y 339.976,Z 828.925,A -85,B 0,C 180,E1 -14318.319,E2 -14318.319} C_VEL
LIN {X 0,Y 340.567,Z 823.867,A -85,B 0,C 180,E1 -14320.101,E2 -14320.101} C_VEL
LIN {X 0,Y 341.385,Z 817.49,A -85,B 0,C 180,E1 -14321.879,E2 -14321.879} C_VEL
LIN {X 0,Y 342.427,Z 809.553,A -85,B 0,C 180,E1 -14323.651,E2 -14323.651} C_VEL
LIN {X 0,Y 343.583,Z 801.433,A -85,B 0,C 180,E1 -14325.116,E2 -14325.116} C_VEL
LIN {X 0,Y 344.705,Z 791.463,A -85,B 0,C 180,E1 -14326.584,E2 -14326.584} C_VEL
LIN {X 0,Y 345.917,Z 780.256,A -85,B 0,C 180,E1 -14327.895,E2 -14327.895} C_VEL
LIN {X 0,Y 347.001,Z 769.249,A -85,B 0,C 180,E1 -14328.907,E2 -14328.907} C_VEL
LIN {X 0,Y 348.045,Z 756.823,A -85,B 0,C 180,E1 -14329.768,E2 -14329.768} C_VEL
LIN {X 0,Y 348.742,Z 743.851,A -85,B 0,C 180,E1 -14330.418,E2 -14330.418} C_VEL
LIN {X 0,Y 349.214,Z 731.236,A -85,B 0,C 180,E1 -14330.813,E2 -14330.813} C_VEL
LIN {X 0,Y 350.198,Z 684.045,A -85,B 0,C 180,E1 -14331.778,E2 -14331.778} C_VEL
LIN {X 0,Y 349.824,Z 678.245,A -85,B 0,C 180,E1 -14331.929,E2 -14331.929} C_VEL
LIN {X 0,Y 347.684,Z 668.861,A -85,B 0,C 180,E1 -14332.278,E2 -14332.278} C_VEL
LIN {X 0,Y 345.599,Z 661.408,A -85,B 0,C 180,E1 -14332.585,E2 -14332.585} C_VEL
LIN {X 0,Y 344.143,Z 653.785,A -85,B 0,C 180,E1 -14332.856,E2 -14332.856} C_VEL
LIN {X 0,Y 339.699,Z 627.914,A -85,B 0,C 180,E1 -14333.76,E2 -14333.76} C_VEL
LIN {X 0,Y 339.136,Z 624.775,A -85,B 0,C 180,E1 -14333.915,E2 -14333.915} C_VEL
LIN {X 0,Y 340.468,Z 605.581,A -85,B 0,C 180,E1 -14337.424,E2 -14337.424} C_VEL
LIN {X 0,Y 341.462,Z 591.451,A -85,B 0,C 180,E1 -14340.18,E2 -14340.18} C_VEL
LIN {X 0,Y 339.051,Z 579.399,A -85,B 0,C 180,E1 -14342.895,E2 -14342.895} C_VEL
LIN {X 0,Y 336.402,Z 568.652,A -85,B 0,C 180,E1 -14345.435,E2 -14345.435} C_VEL
LIN {X 0,Y 333.681,Z 558.928,A -85,B 0,C 180,E1 -14347.788,E2 -14347.788} C_VEL
LIN {X 0,Y 333.642,Z 558.925,A -85,B 0,C 180,E1 -14350.766,E2 -14350.766} C_VEL
LIN {X 0,Y 333.637,Z 558.91,A -85,B 0,C 180,E1 -14354.258,E2 -14354.258} C_VEL
LIN {X 0,Y 333.711,Z 558.916,A -85,B 0,C 180,E1 -14356.12,E2 -14356.12} C_VEL
LIN {X 0,Y 341.206,Z 580.578,A -85,B 0,C 180,E1 -14357.105,E2 -14357.105} C_VEL
LIN {X 0,Y 340.042,Z 634.963,A -85,B 0,C 180,E1 -14358.475,E2 -14358.475} C_VEL
LIN {X 0,Y 339.938,Z 649.261,A -85,B 0,C 180,E1 -14358.998,E2 -14358.998} C_VEL
LIN {X 0,Y 339.574,Z 662.029,A -85,B 0,C 180,E1 -14359.702,E2 -14359.702} C_VEL
LIN {X 0,Y 338.935,Z 674.979,A -85,B 0,C 180,E1 -14360.674,E2 -14360.674} C_VEL
LIN {X 0,Y 338.294,Z 686.664,A -85,B 0,C 180,E1 -14361.81,E2 -14361.81} C_VEL
LIN {X 0,Y 337.482,Z 698.139,A -85,B 0,C 180,E1 -14363.222,E2 -14363.222} C_VEL
LIN {X 0,Y 336.699,Z 707.955,A -85,B 0,C 180,E1 -14364.712,E2 -14364.712} C_VEL
LIN {X 0,Y 335.966,Z 716.49,A -85,B 0,C 180,E1 -14366.308,E2 -14366.308} C_VEL
LIN {X 0,Y 335.317,Z 724.071,A -85,B 0,C 180,E1 -14368.047,E2 -14368.047} C_VEL
LIN {X 0,Y 334.693,Z 731.19,A -85,B 0,C 180,E1 -14370.085,E2 -14370.085} C_VEL
LIN {X 0,Y 334.366,Z 736.268,A -85,B 0,C 180,E1 -14371.977,E2 -14371.977} C_VEL
LIN {X 0,Y 334.075,Z 739.986,A -85,B 0,C 180,E1 -14373.782,E2 -14373.782} C_VEL
LIN {X 0,Y 333.996,Z 742.054,A -85,B 0,C 180,E1 -14375.112,E2 -14375.112} C_VEL
LIN {X 0,Y 333.951,Z 743.61,A -85,B 0,C 180,E1 -14376.431,E2 -14376.431} C_VEL
LIN {X 0,Y 333.987,Z 744.652,A -85,B 0,C 180,E1 -14377.797,E2 -14377.797} C_VEL
LIN {X 0,Y 334.106,Z 745.176,A -85,B 0,C 180,E1 -14379.047,E2 -14379.047} C_VEL
LIN {X 0,Y 334.428,Z 745.056,A -85,B 0,C 180,E1 -14381.022,E2 -14381.022} C_VEL
LIN {X 0,Y 334.907,Z 743.876,A -85,B 0,C 180,E1 -14382.915,E2 -14382.915} C_VEL
LIN {X 0,Y 335.441,Z 742.029,A -85,B 0,C 180,E1 -14384.523,E2 -14384.523} C_VEL
LIN {X 0,Y 336.339,Z 738.229,A -85,B 0,C 180,E1 -14386.712,E2 -14386.712} C_VEL
LIN {X 0,Y 337.343,Z 733.465,A -85,B 0,C 180,E1 -14388.647,E2 -14388.647} C_VEL
LIN {X 0,Y 338.465,Z 727.728,A -85,B 0,C 180,E1 -14390.438,E2 -14390.438} C_VEL
LIN {X 0,Y 339.818,Z 719.985,A -85,B 0,C 180,E1 -14392.334,E2 -14392.334} C_VEL
LIN {X 0,Y 341.258,Z 710.837,A -85,B 0,C 180,E1 -14394.09,E2 -14394.09} C_VEL
LIN {X 0,Y 342.554,Z 701.149,A -85,B 0,C 180,E1 -14395.587,E2 -14395.587} C_VEL
LIN {X 0,Y 343.865,Z 690.181,A -85,B 0,C 180,E1 -14396.925,E2 -14396.925} C_VEL
LIN {X 0,Y 344.82,Z 679.567,A -85,B 0,C 180,E1 -14397.965,E2 -14397.965} C_VEL
LIN {X 0,Y 345.633,Z 668.19,A -85,B 0,C 180,E1 -14398.835,E2 -14398.835} C_VEL
LIN {X 0,Y 346.179,Z 654.56,A -85,B 0,C 180,E1 -14399.605,E2 -14399.605} C_VEL
LIN {X 0,Y 346.36,Z 641.144,A -85,B 0,C 180,E1 -14400.112,E2 -14400.112} C_VEL
LIN {X 0,Y 347.424,Z 606.87,A -85,B 0,C 180,E1 -14401.08,E2 -14401.08} C_VEL
LIN {X 0,Y 348.214,Z 586.285,A -85,B 0,C 180,E1 -14401.66,E2 -14401.66} C_VEL
LIN {X 0,Y 343.264,Z 575.978,A -85,B 0,C 180,E1 -14402.555,E2 -14402.555} C_VEL
LIN {X 0,Y 338.173,Z 566.802,A -85,B 0,C 180,E1 -14403.498,E2 -14403.498} C_VEL
LIN {X 0,Y 335.557,Z 562.726,A -85,B 0,C 180,E1 -14403.978,E2 -14403.978} C_VEL
LIN {X 0,Y 334.033,Z 559.958,A -85,B 0,C 180,E1 -14404.28,E2 -14404.28} C_VEL
LIN {X 0,Y 333.816,Z 558.907,A -85,B 0,C 180,E1 -14404.377,E2 -14404.377} C_VEL
LIN {X 0,Y 334.018,Z 558.874,A -85,B 0,C 180,E1 -14407.253,E2 -14407.253} C_VEL
LIN {X 0,Y 333.827,Z 558.9,A -85,B 0,C 180,E1 -14410.922,E2 -14410.922} C_VEL
LIN {X 0,Y 333.798,Z 558.905,A -85,B 0,C 180,E1 -14414.635,E2 -14414.635} C_VEL
LIN {X 0,Y 333.787,Z 558.908,A -85,B 0,C 180,E1 -14418.656,E2 -14418.656} C_VEL
LIN {X 0,Y 333.683,Z 558.921,A -85,B 0,C 180,E1 -14422.279,E2 -14422.279} C_VEL
LIN {X 0,Y 333.727,Z 558.913,A -85,B 0,C 180,E1 -14426.247,E2 -14426.247} C_VEL
LIN {X 0,Y 333.703,Z 558.917,A -85,B 0,C 180,E1 -14428.973,E2 -14428.973} C_VEL
LIN {X 0,Y 333.635,Z 558.926,A -85,B 0,C 180,E1 -14432.588,E2 -14432.588} C_VEL
LIN {X 0,Y 333.669,Z 558.923,A -85,B 0,C 180,E1 -14436.14,E2 -14436.14} C_VEL
LIN {X 0,Y 333.677,Z 558.922,A -85,B 0,C 180,E1 -14439.188,E2 -14439.188} C_VEL
LIN {X 0,Y 333.697,Z 558.917,A -85,B 0,C 180,E1 -14442.514,E2 -14442.514} C_VEL
LIN {X 0,Y 333.724,Z 558.918,A -85,B 0,C 180,E1 -14445.978,E2 -14445.978} C_VEL
LIN {X 0,Y 333.713,Z 558.988,A -85,B 0,C 180,E1 -14449.368,E2 -14449.368} C_VEL
LIN {X 0,Y 336.67,Z 568.916,A -85,B 0,C 180,E1 -14452.746,E2 -14452.746} C_VEL
LIN {X 0,Y 338.93,Z 577.22,A -85,B 0,C 180,E1 -14455.236,E2 -14455.236} C_VEL
LIN {X 0,Y 341.199,Z 587.468,A -85,B 0,C 180,E1 -14457.988,E2 -14457.988} C_VEL
LIN {X 0,Y 341.963,Z 591.923,A -85,B 0,C 180,E1 -14459.085,E2 -14459.085} C_VEL
LIN {X 0,Y 339.925,Z 605.612,A -85,B 0,C 180,E1 -14461.944,E2 -14461.944} C_VEL
LIN {X 0,Y 338.621,Z 614.934,A -85,B 0,C 180,E1 -14463.832,E2 -14463.832} C_VEL
LIN {X 0,Y 341.952,Z 635.466,A -85,B 0,C 180,E1 -14464.895,E2 -14464.895} C_VEL
LIN {X 0,Y 344.243,Z 654.865,A -85,B 0,C 180,E1 -14465.744,E2 -14465.744} C_VEL
LIN {X 0,Y 345.72,Z 677.868,A -85,B 0,C 180,E1 -14466.598,E2 -14466.598} C_VEL
LIN {X 0,Y 343.693,Z 730.114,A -85,B 0,C 180,E1 -14468.01,E2 -14468.01} C_VEL
LIN {X 0,Y 342.68,Z 743.439,A -85,B 0,C 180,E1 -14468.574,E2 -14468.574} C_VEL
LIN {X 0,Y 341.75,Z 752.146,A -85,B 0,C 180,E1 -14469.066,E2 -14469.066} C_VEL
LIN {X 0,Y 341.124,Z 765.619,A -85,B 0,C 180,E1 -14469.539,E2 -14469.539} C_VEL
LIN {X 0,Y 340.174,Z 778.185,A -85,B 0,C 180,E1 -14470.228,E2 -14470.228} C_VEL
LIN {X 0,Y 339.142,Z 789.886,A -85,B 0,C 180,E1 -14471.109,E2 -14471.109} C_VEL
LIN {X 0,Y 338.006,Z 800.527,A -85,B 0,C 180,E1 -14472.141,E2 -14472.141} C_VEL
LIN {X 0,Y 336.723,Z 811.362,A -85,B 0,C 180,E1 -14473.48,E2 -14473.48} C_VEL
LIN {X 0,Y 335.661,Z 820.18,A -85,B 0,C 180,E1 -14474.829,E2 -14474.829} C_VEL
LIN {X 0,Y 334.656,Z 828.28,A -85,B 0,C 180,E1 -14476.336,E2 -14476.336} C_VEL
LIN {X 0,Y 333.588,Z 836.206,A -85,B 0,C 180,E1 -14478.148,E2 -14478.148} C_VEL
LIN {X 0,Y 333.005,Z 841.557,A -85,B 0,C 180,E1 -14479.667,E2 -14479.667} C_VEL
LIN {X 0,Y 332.506,Z 846.783,A -85,B 0,C 180,E1 -14481.493,E2 -14481.493} C_VEL
LIN {X 0,Y 332.192,Z 850.822,A -85,B 0,C 180,E1 -14483.319,E2 -14483.319} C_VEL
LIN {X 0,Y 332.088,Z 853.8,A -85,B 0,C 180,E1 -14485.145,E2 -14485.145} C_VEL
LIN {X 0,Y 332.073,Z 855.228,A -85,B 0,C 180,E1 -14486.361,E2 -14486.361} C_VEL
LIN {X 0,Y 332.046,Z 856.85,A -85,B 0,C 180,E1 -14488.788,E2 -14488.788} C_VEL
LIN {X 0,Y 332.114,Z 857.07,A -85,B 0,C 180,E1 -14490.001,E2 -14490.001} C_VEL
LIN {X 0,Y 332.028,Z 856.843,A -85,B 0,C 180,E1 -14491.214,E2 -14491.214} C_VEL
LIN {X 0,Y 332.064,Z 855.212,A -85,B 0,C 180,E1 -14493.641,E2 -14493.641} C_VEL
LIN {X 0,Y 332.076,Z 853.775,A -85,B 0,C 180,E1 -14494.857,E2 -14494.857} C_VEL
LIN {X 0,Y 332.187,Z 850.79,A -85,B 0,C 180,E1 -14496.683,E2 -14496.683} C_VEL
LIN {X 0,Y 332.498,Z 846.741,A -85,B 0,C 180,E1 -14498.51,E2 -14498.51} C_VEL
LIN {X 0,Y 333.102,Z 840.492,A -85,B 0,C 180,E1 -14500.639,E2 -14500.639} C_VEL
LIN {X 0,Y 333.865,Z 833.677,A -85,B 0,C 180,E1 -14502.461,E2 -14502.461} C_VEL
LIN {X 0,Y 335.014,Z 825.151,A -85,B 0,C 180,E1 -14504.271,E2 -14504.271} C_VEL
LIN {X 0,Y 336.17,Z 815.486,A -85,B 0,C 180,E1 -14505.912,E2 -14505.912} C_VEL
LIN {X 0,Y 337.344,Z 805.534,A -85,B 0,C 180,E1 -14507.271,E2 -14507.271} C_VEL
LIN {X 0,Y 338.629,Z 794.56,A -85,B 0,C 180,E1 -14508.452,E2 -14508.452} C_VEL
LIN {X 0,Y 339.831,Z 782.255,A -85,B 0,C 180,E1 -14509.481,E2 -14509.481} C_VEL
LIN {X 0,Y 340.744,Z 770.512,A -85,B 0,C 180,E1 -14510.212,E2 -14510.212} C_VEL
LIN {X 0,Y 341.51,Z 757.69,A -85,B 0,C 180,E1 -14510.754,E2 -14510.754} C_VEL
LIN {X 0,Y 342.061,Z 741.292,A -85,B 0,C 180,E1 -14511.152,E2 -14511.152} C_VEL
LIN {X 0,Y 343.106,Z 678.284,A -85,B 0,C 180,E1 -14512.469,E2 -14512.469} C_VEL
LIN {X 0,Y 339.337,Z 644.324,A -85,B 0,C 180,E1 -14513.492,E2 -14513.492} C_VEL
LIN {X 0,Y 338.138,Z 635.775,A -85,B 0,C 180,E1 -14513.789,E2 -14513.789} C_VEL
LIN {X 0,Y 336.611,Z 615.6,A -85,B 0,C 180,E1 -14515.218,E2 -14515.218} C_VEL
LIN {X 0,Y 338.911,Z 593.831,A -85,B 0,C 180,E1 -14519.848,E2 -14519.848} C_VEL
LIN {X 0,Y 339.6,Z 587.701,A -85,B 0,C 180,E1 -14521.157,E2 -14521.157} C_VEL
LIN {X 0,Y 338.825,Z 582.205,A -85,B 0,C 180,E1 -14522.417,E2 -14522.417} C_VEL
LIN {X 0,Y 335.694,Z 567.84,A -85,B 0,C 180,E1 -14525.888,E2 -14525.888} C_VEL
LIN {X 0,Y 333.706,Z 558.918,A -85,B 0,C 180,E1 -14528.122,E2 -14528.122} C_VEL
LIN {X 0,Y 333.649,Z 558.926,A -85,B 0,C 180,E1 -14530.768,E2 -14530.768} C_VEL
LIN {X 0,Y 333.626,Z 558.915,A -85,B 0,C 180,E1 -14534.256,E2 -14534.256} C_VEL
LIN {X 0,Y 333.645,Z 558.915,A -85,B 0,C 180,E1 -14537.619,E2 -14537.619} C_VEL
LIN {X 0,Y 333.655,Z 558.924,A -85,B 0,C 180,E1 -14541.202,E2 -14541.202} C_VEL
LIN {X 0,Y 333.678,Z 558.909,A -85,B 0,C 180,E1 -14543.861,E2 -14543.861} C_VEL
LIN {X 0,Y 333.645,Z 558.917,A -85,B 0,C 180,E1 -14547.413,E2 -14547.413} C_VEL
LIN {X 0,Y 333.712,Z 558.912,A -85,B 0,C 180,E1 -14551.028,E2 -14551.028} C_VEL
LIN {X 0,Y 333.737,Z 558.903,A -85,B 0,C 180,E1 -14553.754,E2 -14553.754} C_VEL
LIN {X 0,Y 333.658,Z 558.923,A -85,B 0,C 180,E1 -14557.719,E2 -14557.719} C_VEL
LIN {X 0,Y 333.795,Z 558.885,A -85,B 0,C 180,E1 -14561.589,E2 -14561.589} C_VEL
LIN {X 0,Y 333.81,Z 558.906,A -85,B 0,C 180,E1 -14565.577,E2 -14565.577} C_VEL
LIN {X 0,Y 333.834,Z 558.88,A -85,B 0,C 180,E1 -14569.078,E2 -14569.078} C_VEL
LIN {X 0,Y 334.008,Z 558.877,A -85,B 0,C 180,E1 -14572.747,E2 -14572.747} C_VEL
LIN {X 0,Y 333.81,Z 558.898,A -85,B 0,C 180,E1 -14575.169,E2 -14575.169} C_VEL
LIN {X 0,Y 334.106,Z 558.844,A -85,B 0,C 180,E1 -14577.589,E2 -14577.589} C_VEL
LIN {X 0,Y 334.228,Z 558.85,A -85,B 0,C 180,E1 -14580,E2 -14580} C_VEL
LIN {X 0,Y 334.106,Z 558.862,A -85,B 0,C 180,E1 -14582.411,E2 -14582.411} C_VEL
LIN {X 0,Y 333.997,Z 558.865,A -85,B 0,C 180,E1 -14586.645,E2 -14586.645} C_VEL
LIN {X 0,Y 333.863,Z 558.897,A -85,B 0,C 180,E1 -14589.695,E2 -14589.695} C_VEL
LIN {X 0,Y 333.798,Z 558.888,A -85,B 0,C 180,E1 -14593.391,E2 -14593.391} C_VEL
LIN {X 0,Y 333.748,Z 558.909,A -85,B 0,C 180,E1 -14597.146,E2 -14597.146} C_VEL
LIN {X 0,Y 333.738,Z 558.895,A -85,B 0,C 180,E1 -14599.69,E2 -14599.69} C_VEL
LIN {X 0,Y 333.694,Z 558.92,A -85,B 0,C 180,E1 -14602.278,E2 -14602.278} C_VEL
LIN {X 0,Y 333.737,Z 558.902,A -85,B 0,C 180,E1 -14606.246,E2 -14606.246} C_VEL
LIN {X 0,Y 333.692,Z 558.916,A -85,B 0,C 180,E1 -14608.974,E2 -14608.974} C_VEL
LIN {X 0,Y 333.648,Z 558.927,A -85,B 0,C 180,E1 -14612.588,E2 -14612.588} C_VEL
LIN {X 0,Y 333.678,Z 558.914,A -85,B 0,C 180,E1 -14616.139,E2 -14616.139} C_VEL
LIN {X 0,Y 333.649,Z 558.92,A -85,B 0,C 180,E1 -14619.192,E2 -14619.192} C_VEL
LIN {X 0,Y 333.635,Z 558.922,A -85,B 0,C 180,E1 -14622.5,E2 -14622.5} C_VEL
LIN {X 0,Y 333.598,Z 558.92,A -85,B 0,C 180,E1 -14625.955,E2 -14625.955} C_VEL
LIN {X 0,Y 333.65,Z 558.923,A -85,B 0,C 180,E1 -14629.315,E2 -14629.315} C_VEL
LIN {X 0,Y 333.668,Z 558.915,A -85,B 0,C 180,E1 -14633.168,E2 -14633.168} C_VEL
LIN {X 0,Y 333.731,Z 559.039,A -85,B 0,C 180,E1 -14633.915,E2 -14633.915} C_VEL
LIN {X 0,Y 337.555,Z 572.634,A -85,B 0,C 180,E1 -14636.883,E2 -14636.883} C_VEL
LIN {X 0,Y 340.309,Z 583.829,A -85,B 0,C 180,E1 -14639.227,E2 -14639.227} C_VEL
LIN {X 0,Y 342.097,Z 593.328,A -85,B 0,C 180,E1 -14641.132,E2 -14641.132} C_VEL
LIN {X 0,Y 340.418,Z 614.025,A -85,B 0,C 180,E1 -14644.634,E2 -14644.634} C_VEL
LIN {X 0,Y 339.884,Z 624.554,A -85,B 0,C 180,E1 -14646.285,E2 -14646.285} C_VEL
LIN {X 0,Y 344.149,Z 651.06,A -85,B 0,C 180,E1 -14647.19,E2 -14647.19} C_VEL
LIN {X 0,Y 342.465,Z 735.774,A -85,B 0,C 180,E1 -14648.992,E2 -14648.992} C_VEL
LIN {X 0,Y 341.801,Z 749.14,A -85,B 0,C 180,E1 -14649.5,E2 -14649.5} C_VEL
LIN {X 0,Y 340.836,Z 762.206,A -85,B 0,C 180,E1 -14650.265,E2 -14650.265} C_VEL
LIN {X 0,Y 339.917,Z 773.34,A -85,B 0,C 180,E1 -14651.151,E2 -14651.151} C_VEL
LIN {X 0,Y 338.746,Z 783.866,A -85,B 0,C 180,E1 -14652.211,E2 -14652.211} C_VEL
LIN {X 0,Y 337.631,Z 794.359,A -85,B 0,C 180,E1 -14653.556,E2 -14653.556} C_VEL
LIN {X 0,Y 336.283,Z 804.491,A -85,B 0,C 180,E1 -14655.166,E2 -14655.166} C_VEL
LIN {X 0,Y 335.165,Z 812.126,A -85,B 0,C 180,E1 -14656.663,E2 -14656.663} C_VEL
LIN {X 0,Y 334.17,Z 819.569,A -85,B 0,C 180,E1 -14658.474,E2 -14658.474} C_VEL
LIN {X 0,Y 333.356,Z 825.548,A -85,B 0,C 180,E1 -14660.289,E2 -14660.289} C_VEL
LIN {X 0,Y 332.807,Z 830.272,A -85,B 0,C 180,E1 -14662.11,E2 -14662.11} C_VEL
LIN {X 0,Y 332.429,Z 833.884,A -85,B 0,C 180,E1 -14663.931,E2 -14663.931} C_VEL
LIN {X 0,Y 332.266,Z 835.743,A -85,B 0,C 180,E1 -14665.146,E2 -14665.146} C_VEL
LIN {X 0,Y 332.112,Z 837.165,A -85,B 0,C 180,E1 -14666.359,E2 -14666.359} C_VEL
LIN {X 0,Y 331.963,Z 838.775,A -85,B 0,C 180,E1 -14668.786,E2 -14668.786} C_VEL
LIN {X 0,Y 331.973,Z 839.008,A -85,B 0,C 180,E1 -14669.999,E2 -14669.999} C_VEL
LIN {X 0,Y 331.962,Z 838.816,A -85,B 0,C 180,E1 -14671.212,E2 -14671.212} C_VEL
LIN {X 0,Y 332.105,Z 837.262,A -85,B 0,C 180,E1 -14673.639,E2 -14673.639} C_VEL
LIN {X 0,Y 332.263,Z 835.895,A -85,B 0,C 180,E1 -14674.852,E2 -14674.852} C_VEL
LIN {X 0,Y 332.522,Z 833.153,A -85,B 0,C 180,E1 -14676.601,E2 -14676.601} C_VEL
LIN {X 0,Y 332.93,Z 829.116,A -85,B 0,C 180,E1 -14678.496,E2 -14678.496} C_VEL
LIN {X 0,Y 333.575,Z 824.056,A -85,B 0,C 180,E1 -14680.315,E2 -14680.315} C_VEL
LIN {X 0,Y 334.449,Z 817.677,A -85,B 0,C 180,E1 -14682.129,E2 -14682.129} C_VEL
LIN {X 0,Y 335.523,Z 809.739,A -85,B 0,C 180,E1 -14683.937,E2 -14683.937} C_VEL
LIN {X 0,Y 336.743,Z 801.616,A -85,B 0,C 180,E1 -14685.431,E2 -14685.431} C_VEL
LIN {X 0,Y 337.912,Z 791.642,A -85,B 0,C 180,E1 -14686.927,E2 -14686.927} C_VEL
LIN {X 0,Y 339.17,Z 780.43,A -85,B 0,C 180,E1 -14688.263,E2 -14688.263} C_VEL
LIN {X 0,Y 340.311,Z 769.415,A -85,B 0,C 180,E1 -14689.293,E2 -14689.293} C_VEL
LIN {X 0,Y 341.381,Z 756.976,A -85,B 0,C 180,E1 -14690.17,E2 -14690.17} C_VEL
LIN {X 0,Y 342.053,Z 744.822,A -85,B 0,C 180,E1 -14690.796,E2 -14690.796} C_VEL
LIN {X 0,Y 342.579,Z 732.827,A -85,B 0,C 180,E1 -14691.196,E2 -14691.196} C_VEL
LIN {X 0,Y 344.143,Z 653.785,A -85,B 0,C 180,E1 -14692.856,E2 -14692.856} C_VEL
LIN {X 0,Y 342.777,Z 648.201,A -85,B 0,C 180,E1 -14693.079,E2 -14693.079} C_VEL
LIN {X 0,Y 338.538,Z 639.71,A -85,B 0,C 180,E1 -14693.577,E2 -14693.577} C_VEL
LIN {X 0,Y 334.154,Z 631.268,A -85,B 0,C 180,E1 -14694.102,E2 -14694.102} C_VEL
LIN {X 0,Y 332.548,Z 625.746,A -85,B 0,C 180,E1 -14694.356,E2 -14694.356} C_VEL
LIN {X 0,Y 332.462,Z 625.029,A -85,B 0,C 180,E1 -14694.406,E2 -14694.406} C_VEL
LIN {X 0,Y 333.786,Z 606.504,A -85,B 0,C 180,E1 -14697.831,E2 -14697.831} C_VEL
LIN {X 0,Y 334.762,Z 594.14,A -85,B 0,C 180,E1 -14700.254,E2 -14700.254} C_VEL
LIN {X 0,Y 333.353,Z 585.93,A -85,B 0,C 180,E1 -14702.103,E2 -14702.103} C_VEL
LIN {X 0,Y 330.452,Z 573.514,A -85,B 0,C 180,E1 -14705.044,E2 -14705.044} C_VEL
LIN {X 0,Y 326.975,Z 561.153,A -85,B 0,C 180,E1 -14708.06,E2 -14708.06} C_VEL
LIN {X 0,Y 326.63,Z 559.795,A -85,B 0,C 180,E1 -14708.426,E2 -14708.426} C_VEL
LIN {X 0,Y 326.572,Z 559.804,A -85,B 0,C 180,E1 -14711.844,E2 -14711.844} C_VEL
LIN {X 0,Y 326.676,Z 559.977,A -85,B 0,C 180,E1 -14715.785,E2 -14715.785} C_VEL
LIN {X 0,Y 334.233,Z 581.146,A -85,B 0,C 180,E1 -14716.777,E2 -14716.777} C_VEL
LIN {X 0,Y 333.13,Z 640.85,A -85,B 0,C 180,E1 -14718.352,E2 -14718.352} C_VEL
LIN {X 0,Y 332.93,Z 654.938,A -85,B 0,C 180,E1 -14718.976,E2 -14718.976} C_VEL
LIN {X 0,Y 332.453,Z 667.379,A -85,B 0,C 180,E1 -14719.757,E2 -14719.757} C_VEL
LIN {X 0,Y 331.863,Z 679.172,A -85,B 0,C 180,E1 -14720.743,E2 -14720.743} C_VEL
LIN {X 0,Y 331.134,Z 691.128,A -85,B 0,C 180,E1 -14722.012,E2 -14722.012} C_VEL
LIN {X 0,Y 330.286,Z 701.797,A -85,B 0,C 180,E1 -14723.43,E2 -14723.43} C_VEL
LIN {X 0,Y 329.431,Z 712.474,A -85,B 0,C 180,E1 -14725.202,E2 -14725.202} C_VEL
LIN {X 0,Y 328.656,Z 720.94,A -85,B 0,C 180,E1 -14726.955,E2 -14726.955} C_VEL
LIN {X 0,Y 327.907,Z 728.995,A -85,B 0,C 180,E1 -14729.043,E2 -14729.043} C_VEL
LIN {X 0,Y 327.462,Z 735.162,A -85,B 0,C 180,E1 -14731.111,E2 -14731.111} C_VEL
LIN {X 0,Y 327.122,Z 739.844,A -85,B 0,C 180,E1 -14733.181,E2 -14733.181} C_VEL
LIN {X 0,Y 326.987,Z 742.219,A -85,B 0,C 180,E1 -14734.541,E2 -14734.541} C_VEL
LIN {X 0,Y 326.928,Z 743.988,A -85,B 0,C 180,E1 -14735.893,E2 -14735.893} C_VEL
LIN {X 0,Y 326.966,Z 745.499,A -85,B 0,C 180,E1 -14737.553,E2 -14737.553} C_VEL
LIN {X 0,Y 327.209,Z 746.318,A -85,B 0,C 180,E1 -14739.9,E2 -14739.9} C_VEL
LIN {X 0,Y 327.477,Z 746.14,A -85,B 0,C 180,E1 -14741.221,E2 -14741.221} C_VEL
LIN {X 0,Y 327.802,Z 745.439,A -85,B 0,C 180,E1 -14742.533,E2 -14742.533} C_VEL
LIN {X 0,Y 328.389,Z 743.674,A -85,B 0,C 180,E1 -14744.372,E2 -14744.372} C_VEL
LIN {X 0,Y 329.234,Z 740.516,A -85,B 0,C 180,E1 -14746.419,E2 -14746.419} C_VEL
LIN {X 0,Y 330.182,Z 736.51,A -85,B 0,C 180,E1 -14748.262,E2 -14748.262} C_VEL
LIN {X 0,Y 331.406,Z 730.866,A -85,B 0,C 180,E1 -14750.232,E2 -14750.232} C_VEL
LIN {X 0,Y 332.817,Z 723.647,A -85,B 0,C 180,E1 -14752.172,E2 -14752.172} C_VEL
LIN {X 0,Y 334.294,Z 715.206,A -85,B 0,C 180,E1 -14753.966,E2 -14753.966} C_VEL
LIN {X 0,Y 335.63,Z 706.225,A -85,B 0,C 180,E1 -14755.496,E2 -14755.496} C_VEL
LIN {X 0,Y 336.964,Z 696.226,A -85,B 0,C 180,E1 -14756.862,E2 -14756.862} C_VEL
LIN {X 0,Y 338.189,Z 685.214,A -85,B 0,C 180,E1 -14758.069,E2 -14758.069} C_VEL
LIN {X 0,Y 339.182,Z 673.061,A -85,B 0,C 180,E1 -14759.11,E2 -14759.11} C_VEL
LIN {X 0,Y 339.871,Z 660.507,A -85,B 0,C 180,E1 -14759.926,E2 -14759.926} C_VEL
LIN {X 0,Y 340.229,Z 647.921,A -85,B 0,C 180,E1 -14760.501,E2 -14760.501} C_VEL
LIN {X 0,Y 340.78,Z 622.633,A -85,B 0,C 180,E1 -14761.273,E2 -14761.273} C_VEL
LIN {X 0,Y 342.163,Z 588.474,A -85,B 0,C 180,E1 -14762.257,E2 -14762.257} C_VEL
LIN {X 0,Y 338.074,Z 579.9,A -85,B 0,C 180,E1 -14763.04,E2 -14763.04} C_VEL
LIN {X 0,Y 333.171,Z 571.13,A -85,B 0,C 180,E1 -14763.982,E2 -14763.982} C_VEL
LIN {X 0,Y 329.221,Z 564.429,A -85,B 0,C 180,E1 -14764.779,E2 -14764.779} C_VEL
LIN {X 0,Y 327.334,Z 561.652,A -85,B 0,C 180,E1 -14765.158,E2 -14765.158} C_VEL
LIN {X 0,Y 326.828,Z 559.771,A -85,B 0,C 180,E1 -14765.321,E2 -14765.321} C_VEL
LIN {X 0,Y 326.971,Z 559.751,A -85,B 0,C 180,E1 -14767.41,E2 -14767.41} C_VEL
LIN {X 0,Y 326.763,Z 559.783,A -85,B 0,C 180,E1 -14771.161,E2 -14771.161} C_VEL
LIN {X 0,Y 326.744,Z 559.78,A -85,B 0,C 180,E1 -14774.958,E2 -14774.958} C_VEL
LIN {X 0,Y 326.724,Z 559.79,A -85,B 0,C 180,E1 -14778.839,E2 -14778.839} C_VEL
LIN {X 0,Y 326.612,Z 559.8,A -85,B 0,C 180,E1 -14782.788,E2 -14782.788} C_VEL
LIN {X 0,Y 326.681,Z 559.791,A -85,B 0,C 180,E1 -14785.485,E2 -14785.485} C_VEL
LIN {X 0,Y 326.652,Z 559.795,A -85,B 0,C 180,E1 -14789.66,E2 -14789.66} C_VEL
LIN {X 0,Y 326.599,Z 559.799,A -85,B 0,C 180,E1 -14794.02,E2 -14794.02} C_VEL
LIN {X 0,Y 326.622,Z 559.794,A -85,B 0,C 180,E1 -14797.24,E2 -14797.24} C_VEL
LIN {X 0,Y 326.629,Z 559.795,A -85,B 0,C 180,E1 -14800.204,E2 -14800.204} C_VEL
LIN {X 0,Y 326.652,Z 559.797,A -85,B 0,C 180,E1 -14803.511,E2 -14803.511} C_VEL
LIN {X 0,Y 326.645,Z 559.795,A -85,B 0,C 180,E1 -14807.015,E2 -14807.015} C_VEL
LIN {X 0,Y 326.647,Z 559.904,A -85,B 0,C 180,E1 -14808.317,E2 -14808.317} C_VEL
LIN {X 0,Y 329.266,Z 568.249,A -85,B 0,C 180,E1 -14811.404,E2 -14811.404} C_VEL
LIN {X 0,Y 331.907,Z 577.76,A -85,B 0,C 180,E1 -14814.441,E2 -14814.441} C_VEL
LIN {X 0,Y 334.155,Z 587.792,A -85,B 0,C 180,E1 -14817.276,E2 -14817.276} C_VEL
LIN {X 0,Y 335.233,Z 594.48,A -85,B 0,C 180,E1 -14818.999,E2 -14818.999} C_VEL
LIN {X 0,Y 332.21,Z 613.416,A -85,B 0,C 180,E1 -14823.001,E2 -14823.001} C_VEL
LIN {X 0,Y 335.425,Z 632.828,A -85,B 0,C 180,E1 -14824.085,E2 -14824.085} C_VEL
LIN {X 0,Y 337.653,Z 650.828,A -85,B 0,C 180,E1 -14824.933,E2 -14824.933} C_VEL
LIN {X 0,Y 339.147,Z 671.106,A -85,B 0,C 180,E1 -14825.755,E2 -14825.755} C_VEL
LIN {X 0,Y 339.442,Z 680.589,A -85,B 0,C 180,E1 -14826.083,E2 -14826.083} C_VEL
LIN {X 0,Y 337.484,Z 728.972,A -85,B 0,C 180,E1 -14827.423,E2 -14827.423} C_VEL
LIN {X 0,Y 336.388,Z 742.18,A -85,B 0,C 180,E1 -14827.992,E2 -14827.992} C_VEL
LIN {X 0,Y 335.025,Z 754.763,A -85,B 0,C 180,E1 -14828.706,E2 -14828.706} C_VEL
LIN {X 0,Y 334.302,Z 767.721,A -85,B 0,C 180,E1 -14829.223,E2 -14829.223} C_VEL
LIN {X 0,Y 333.314,Z 780.252,A -85,B 0,C 180,E1 -14829.964,E2 -14829.964} C_VEL
LIN {X 0,Y 332.253,Z 791.425,A -85,B 0,C 180,E1 -14830.862,E2 -14830.862} C_VEL
LIN {X 0,Y 330.912,Z 802.946,A -85,B 0,C 180,E1 -14832.065,E2 -14832.065} C_VEL
LIN {X 0,Y 329.656,Z 813.307,A -85,B 0,C 180,E1 -14833.435,E2 -14833.435} C_VEL
LIN {X 0,Y 328.526,Z 821.902,A -85,B 0,C 180,E1 -14834.833,E2 -14834.833} C_VEL
LIN {X 0,Y 327.533,Z 829.565,A -85,B 0,C 180,E1 -14836.349,E2 -14836.349} C_VEL
LIN {X 0,Y 326.461,Z 837.146,A -85,B 0,C 180,E1 -14838.2,E2 -14838.2} C_VEL
LIN {X 0,Y 325.798,Z 843.231,A -85,B 0,C 180,E1 -14840.064,E2 -14840.064} C_VEL
LIN {X 0,Y 325.31,Z 848.039,A -85,B 0,C 180,E1 -14841.929,E2 -14841.929} C_VEL
LIN {X 0,Y 325.042,Z 852.146,A -85,B 0,C 180,E1 -14844.047,E2 -14844.047} C_VEL
LIN {X 0,Y 324.998,Z 855.036,A -85,B 0,C 180,E1 -14846.281,E2 -14846.281} C_VEL
LIN {X 0,Y 324.949,Z 856.657,A -85,B 0,C 180,E1 -14848.762,E2 -14848.762} C_VEL
LIN {X 0,Y 325.016,Z 856.877,A -85,B 0,C 180,E1 -14850.001,E2 -14850.001} C_VEL
LIN {X 0,Y 324.924,Z 856.03,A -85,B 0,C 180,E1 -14852.48,E2 -14852.48} C_VEL
LIN {X 0,Y 324.989,Z 855.019,A -85,B 0,C 180,E1 -14853.721,E2 -14853.721} C_VEL
LIN {X 0,Y 325.019,Z 852.185,A -85,B 0,C 180,E1 -14855.914,E2 -14855.914} C_VEL
LIN {X 0,Y 325.344,Z 848,A -85,B 0,C 180,E1 -14858.073,E2 -14858.073} C_VEL
LIN {X 0,Y 325.784,Z 843.179,A -85,B 0,C 180,E1 -14859.939,E2 -14859.939} C_VEL
LIN {X 0,Y 326.424,Z 837.076,A -85,B 0,C 180,E1 -14861.803,E2 -14861.803} C_VEL
LIN {X 0,Y 327.504,Z 829.48,A -85,B 0,C 180,E1 -14863.654,E2 -14863.654} C_VEL
LIN {X 0,Y 328.716,Z 820.326,A -85,B 0,C 180,E1 -14865.426,E2 -14865.426} C_VEL
LIN {X 0,Y 329.908,Z 810.209,A -85,B 0,C 180,E1 -14867.001,E2 -14867.001} C_VEL
LIN {X 0,Y 331.208,Z 800.188,A -85,B 0,C 180,E1 -14868.24,E2 -14868.24} C_VEL
LIN {X 0,Y 332.424,Z 789.514,A -85,B 0,C 180,E1 -14869.29,E2 -14869.29} C_VEL
LIN {X 0,Y 333.559,Z 776.654,A -85,B 0,C 180,E1 -14870.264,E2 -14870.264} C_VEL
LIN {X 0,Y 334.481,Z 764.224,A -85,B 0,C 180,E1 -14870.929,E2 -14870.929} C_VEL
LIN {X 0,Y 335.154,Z 751.329,A -85,B 0,C 180,E1 -14871.368,E2 -14871.368} C_VEL
LIN {X 0,Y 336.586,Z 679.547,A -85,B 0,C 180,E1 -14872.898,E2 -14872.898} C_VEL
LIN {X 0,Y 333.068,Z 646.962,A -85,B 0,C 180,E1 -14873.899,E2 -14873.899} C_VEL
LIN {X 0,Y 331.516,Z 635.999,A -85,B 0,C 180,E1 -14874.275,E2 -14874.275} C_VEL
LIN {X 0,Y 329.808,Z 613.565,A -85,B 0,C 180,E1 -14875.903,E2 -14875.903} C_VEL
LIN {X 0,Y 332.068,Z 593.411,A -85,B 0,C 180,E1 -14880.279,E2 -14880.279} C_VEL
LIN {X 0,Y 332.619,Z 587.718,A -85,B 0,C 180,E1 -14881.531,E2 -14881.531} C_VEL
LIN {X 0,Y 330.161,Z 575.578,A -85,B 0,C 180,E1 -14884.467,E2 -14884.467} C_VEL
LIN {X 0,Y 326.975,Z 561.352,A -85,B 0,C 180,E1 -14888.061,E2 -14888.061} C_VEL
LIN {X 0,Y 326.622,Z 559.802,A -85,B 0,C 180,E1 -14888.522,E2 -14888.522} C_VEL
LIN {X 0,Y 326.578,Z 559.805,A -85,B 0,C 180,E1 -14891.846,E2 -14891.846} C_VEL
LIN {X 0,Y 326.559,Z 559.804,A -85,B 0,C 180,E1 -14895.252,E2 -14895.252} C_VEL
LIN {X 0,Y 326.58,Z 559.793,A -85,B 0,C 180,E1 -14898.869,E2 -14898.869} C_VEL
LIN {X 0,Y 326.63,Z 559.787,A -85,B 0,C 180,E1 -14902.762,E2 -14902.762} C_VEL
LIN {X 0,Y 326.609,Z 559.8,A -85,B 0,C 180,E1 -14905.981,E2 -14905.981} C_VEL
LIN {X 0,Y 326.662,Z 559.787,A -85,B 0,C 180,E1 -14910.341,E2 -14910.341} C_VEL
LIN {X 0,Y 326.691,Z 559.776,A -85,B 0,C 180,E1 -14914.516,E2 -14914.516} C_VEL
LIN {X 0,Y 326.621,Z 559.798,A -85,B 0,C 180,E1 -14918.544,E2 -14918.544} C_VEL
LIN {X 0,Y 326.746,Z 559.767,A -85,B 0,C 180,E1 -14921.178,E2 -14921.178} C_VEL
LIN {X 0,Y 326.764,Z 559.782,A -85,B 0,C 180,E1 -14925.433,E2 -14925.433} C_VEL
LIN {X 0,Y 326.771,Z 559.761,A -85,B 0,C 180,E1 -14928.839,E2 -14928.839} C_VEL
LIN {X 0,Y 326.96,Z 559.754,A -85,B 0,C 180,E1 -14932.59,E2 -14932.59} C_VEL
LIN {X 0,Y 326.777,Z 559.776,A -85,B 0,C 180,E1 -14935.065,E2 -14935.065} C_VEL
LIN {X 0,Y 327.046,Z 559.722,A -85,B 0,C 180,E1 -14937.537,E2 -14937.537} C_VEL
LIN {X 0,Y 327.18,Z 559.728,A -85,B 0,C 180,E1 -14940,E2 -14940} C_VEL
LIN {X 0,Y 327.047,Z 559.741,A -85,B 0,C 180,E1 -14942.463,E2 -14942.463} C_VEL
LIN {X 0,Y 326.965,Z 559.741,A -85,B 0,C 180,E1 -14946.638,E2 -14946.638} C_VEL
LIN {X 0,Y 326.814,Z 559.772,A -85,B 0,C 180,E1 -14949.906,E2 -14949.906} C_VEL
LIN {X 0,Y 326.76,Z 559.766,A -85,B 0,C 180,E1 -14953.685,E2 -14953.685} C_VEL
LIN {X 0,Y 326.701,Z 559.783,A -85,B 0,C 180,E1 -14957.528,E2 -14957.528} C_VEL
LIN {X 0,Y 326.664,Z 559.779,A -85,B 0,C 180,E1 -14960.135,E2 -14960.135} C_VEL
LIN {X 0,Y 326.654,Z 559.785,A -85,B 0,C 180,E1 -14964.129,E2 -14964.129} C_VEL
LIN {X 0,Y 326.684,Z 559.788,A -85,B 0,C 180,E1 -14966.858,E2 -14966.858} C_VEL
LIN {X 0,Y 326.636,Z 559.785,A -85,B 0,C 180,E1 -14970.61,E2 -14970.61} C_VEL
LIN {X 0,Y 326.61,Z 559.801,A -85,B 0,C 180,E1 -14974.019,E2 -14974.019} C_VEL
LIN {X 0,Y 326.629,Z 559.8,A -85,B 0,C 180,E1 -14977.238,E2 -14977.238} C_VEL
LIN {X 0,Y 326.58,Z 559.806,A -85,B 0,C 180,E1 -14981.131,E2 -14981.131} C_VEL
LIN {X 0,Y 326.53,Z 559.812,A -85,B 0,C 180,E1 -14984.743,E2 -14984.743} C_VEL
LIN {X 0,Y 326.578,Z 559.784,A -85,B 0,C 180,E1 -14988.154,E2 -14988.154} C_VEL
LIN {X 0,Y 326.601,Z 559.79,A -85,B 0,C 180,E1 -14991.388,E2 -14991.388} C_VEL
LIN {X 0,Y 326.675,Z 559.954,A -85,B 0,C 180,E1 -14993.295,E2 -14993.295} C_VEL
LIN {X 0,Y 330.275,Z 572.356,A -85,B 0,C 180,E1 -14996.088,E2 -14996.088} C_VEL
LIN {X 0,Y 333.58,Z 585.606,A -85,B 0,C 180,E1 -14998.924,E2 -14998.924} C_VEL
LIN {X 0,Y 335.407,Z 595.08,A -85,B 0,C 180,E1 -15000.844,E2 -15000.844} C_VEL
LIN {X 0,Y 333.678,Z 616.023,A -85,B 0,C 180,E1 -15004.42,E2 -15004.42} C_VEL
LIN {X 0,Y 333.206,Z 624.362,A -85,B 0,C 180,E1 -15005.773,E2 -15005.773} C_VEL
LIN {X 0,Y 337.642,Z 652.242,A -85,B 0,C 180,E1 -15006.75,E2 -15006.75} C_VEL
LIN {X 0,Y 335.862,Z 735.904,A -85,B 0,C 180,E1 -15008.559,E2 -15008.559} C_VEL
LIN {X 0,Y 335.186,Z 749.303,A -85,B 0,C 180,E1 -15009.077,E2 -15009.077} C_VEL
LIN {X 0,Y 334.185,Z 762.38,A -85,B 0,C 180,E1 -15009.856,E2 -15009.856} C_VEL
LIN {X 0,Y 333.211,Z 773.52,A -85,B 0,C 180,E1 -15010.757,E2 -15010.757} C_VEL
LIN {X 0,Y 332.009,Z 783.787,A -85,B 0,C 180,E1 -15011.806,E2 -15011.806} C_VEL
LIN {X 0,Y 330.925,Z 793.679,A -85,B 0,C 180,E1 -15013.08,E2 -15013.08} C_VEL
LIN {X 0,Y 329.663,Z 802.948,A -85,B 0,C 180,E1 -15014.544,E2 -15014.544} C_VEL
LIN {X 0,Y 328.259,Z 812.317,A -85,B 0,C 180,E1 -15016.378,E2 -15016.378} C_VEL
LIN {X 0,Y 327.206,Z 819.762,A -85,B 0,C 180,E1 -15018.225,E2 -15018.225} C_VEL
LIN {X 0,Y 326.356,Z 825.741,A -85,B 0,C 180,E1 -15020.079,E2 -15020.079} C_VEL
LIN {X 0,Y 325.758,Z 830.466,A -85,B 0,C 180,E1 -15021.938,E2 -15021.938} C_VEL
LIN {X 0,Y 325.371,Z 834.077,A -85,B 0,C 180,E1 -15023.799,E2 -15023.799} C_VEL
LIN {X 0,Y 325.193,Z 835.937,A -85,B 0,C 180,E1 -15025.04,E2 -15025.04} C_VEL
LIN {X 0,Y 325.044,Z 837.358,A -85,B 0,C 180,E1 -15026.28,E2 -15026.28} C_VEL
LIN {X 0,Y 324.871,Z 838.968,A -85,B 0,C 180,E1 -15028.759,E2 -15028.759} C_VEL
LIN {X 0,Y 324.878,Z 839.201,A -85,B 0,C 180,E1 -15029.999,E2 -15029.999} C_VEL
LIN {X 0,Y 324.87,Z 839.009,A -85,B 0,C 180,E1 -15031.239,E2 -15031.239} C_VEL
LIN {X 0,Y 325.038,Z 837.454,A -85,B 0,C 180,E1 -15033.718,E2 -15033.718} C_VEL
LIN {X 0,Y 325.189,Z 836.087,A -85,B 0,C 180,E1 -15034.958,E2 -15034.958} C_VEL
LIN {X 0,Y 325.448,Z 833.582,A -85,B 0,C 180,E1 -15036.602,E2 -15036.602} C_VEL
LIN {X 0,Y 325.895,Z 829.306,A -85,B 0,C 180,E1 -15038.681,E2 -15038.681} C_VEL
LIN {X 0,Y 326.595,Z 824.245,A -85,B 0,C 180,E1 -15040.538,E2 -15040.538} C_VEL
LIN {X 0,Y 327.494,Z 817.865,A -85,B 0,C 180,E1 -15042.391,E2 -15042.391} C_VEL
LIN {X 0,Y 328.637,Z 809.925,A -85,B 0,C 180,E1 -15044.236,E2 -15044.236} C_VEL
LIN {X 0,Y 329.908,Z 801.799,A -85,B 0,C 180,E1 -15045.759,E2 -15045.759} C_VEL
LIN {X 0,Y 331.12,Z 791.822,A -85,B 0,C 180,E1 -15047.285,E2 -15047.285} C_VEL
LIN {X 0,Y 332.429,Z 780.604,A -85,B 0,C 180,E1 -15048.647,E2 -15048.647} C_VEL
LIN {X 0,Y 333.639,Z 769.581,A -85,B 0,C 180,E1 -15049.695,E2 -15049.695} C_VEL
LIN {X 0,Y 334.741,Z 757.128,A -85,B 0,C 180,E1 -15050.588,E2 -15050.588} C_VEL
LIN {X 0,Y 335.438,Z 744.954,A -85,B 0,C 180,E1 -15051.226,E2 -15051.226} C_VEL
LIN {X 0,Y 335.987,Z 732.915,A -85,B 0,C 180,E1 -15051.632,E2 -15051.632} C_VEL
LIN {X 0,Y 337.583,Z 654.437,A -85,B 0,C 180,E1 -15053.312,E2 -15053.312} C_VEL
LIN {X 0,Y 333.414,Z 630.062,A -85,B 0,C 180,E1 -15054.187,E2 -15054.187} C_VEL
LIN {X 0,Y 332.548,Z 625.746,A -85,B 0,C 180,E1 -15054.356,E2 -15054.356} C_VEL
LIN {X 0,Y 332.036,Z 624.464,A -85,B 0,C 180,E1 -15054.546,E2 -15054.546} C_VEL
LIN {X 0,Y 328.963,Z 617.628,A -85,B 0,C 180,E1 -15056.075,E2 -15056.075} C_VEL
LIN {X 0,Y 327.317,Z 611.431,A -85,B 0,C 180,E1 -15057.495,E2 -15057.495} C_VEL
LIN {X 0,Y 327.243,Z 605.972,A -85,B 0,C 180,E1 -15058.537,E2 -15058.537} C_VEL
LIN {X 0,Y 328.046,Z 595.328,A -85,B 0,C 180,E1 -15060.657,E2 -15060.657} C_VEL
LIN {X 0,Y 325.74,Z 583.637,A -85,B 0,C 180,E1 -15063.376,E2 -15063.376} C_VEL
LIN {X 0,Y 322.709,Z 571.454,A -85,B 0,C 180,E1 -15066.313,E2 -15066.313} C_VEL
LIN {X 0,Y 319.578,Z 560.667,A -85,B 0,C 180,E1 -15069.104,E2 -15069.104} C_VEL
LIN {X 0,Y 319.559,Z 560.659,A -85,B 0,C 180,E1 -15073.467,E2 -15073.467} C_VEL
LIN {X 0,Y 319.596,Z 560.817,A -85,B 0,C 180,E1 -15075.414,E2 -15075.414} C_VEL
LIN {X 0,Y 327.49,Z 582.833,A -85,B 0,C 180,E1 -15076.478,E2 -15076.478} C_VEL
LIN {X 0,Y 326.313,Z 637.689,A -85,B 0,C 180,E1 -15077.941,E2 -15077.941} C_VEL
LIN {X 0,Y 326.15,Z 651.953,A -85,B 0,C 180,E1 -15078.5,E2 -15078.5} C_VEL
LIN {X 0,Y 325.712,Z 664.911,A -85,B 0,C 180,E1 -15079.266,E2 -15079.266} C_VEL
LIN {X 0,Y 325.08,Z 677.6,A -85,B 0,C 180,E1 -15080.273,E2 -15080.273} C_VEL
LIN {X 0,Y 324.371,Z 689.244,A -85,B 0,C 180,E1 -15081.471,E2 -15081.471} C_VEL
LIN {X 0,Y 323.523,Z 700.185,A -85,B 0,C 180,E1 -15082.876,E2 -15082.876} C_VEL
LIN {X 0,Y 322.755,Z 709.688,A -85,B 0,C 180,E1 -15084.375,E2 -15084.375} C_VEL
LIN {X 0,Y 321.954,Z 718.341,A -85,B 0,C 180,E1 -15086.045,E2 -15086.045} C_VEL
LIN {X 0,Y 321.239,Z 726.361,A -85,B 0,C 180,E1 -15087.958,E2 -15087.958} C_VEL
LIN {X 0,Y 320.615,Z 733.438,A -85,B 0,C 180,E1 -15090.087,E2 -15090.087} C_VEL
LIN {X 0,Y 320.299,Z 738.225,A -85,B 0,C 180,E1 -15091.939,E2 -15091.939} C_VEL
LIN {X 0,Y 319.968,Z 742.65,A -85,B 0,C 180,E1 -15094.226,E2 -15094.226} C_VEL
LIN {X 0,Y 319.898,Z 744.257,A -85,B 0,C 180,E1 -15095.328,E2 -15095.328} C_VEL
LIN {X 0,Y 319.925,Z 746.301,A -85,B 0,C 180,E1 -15097.311,E2 -15097.311} C_VEL
LIN {X 0,Y 320.122,Z 747.349,A -85,B 0,C 180,E1 -15099.435,E2 -15099.435} C_VEL
LIN {X 0,Y 320.361,Z 747.36,A -85,B 0,C 180,E1 -15100.788,E2 -15100.788} C_VEL
LIN {X 0,Y 320.685,Z 746.923,A -85,B 0,C 180,E1 -15102.132,E2 -15102.132} C_VEL
LIN {X 0,Y 321.361,Z 745.296,A -85,B 0,C 180,E1 -15104.201,E2 -15104.201} C_VEL
LIN {X 0,Y 322.455,Z 741.563,A -85,B 0,C 180,E1 -15106.77,E2 -15106.77} C_VEL
LIN {X 0,Y 323.492,Z 737.395,A -85,B 0,C 180,E1 -15108.724,E2 -15108.724} C_VEL
LIN {X 0,Y 324.771,Z 731.935,A -85,B 0,C 180,E1 -15110.66,E2 -15110.66} C_VEL
LIN {X 0,Y 326.218,Z 724.952,A -85,B 0,C 180,E1 -15112.573,E2 -15112.573} C_VEL
LIN {X 0,Y 327.868,Z 716.197,A -85,B 0,C 180,E1 -15114.465,E2 -15114.465} C_VEL
LIN {X 0,Y 329.419,Z 706.154,A -85,B 0,C 180,E1 -15116.177,E2 -15116.177} C_VEL
LIN {X 0,Y 330.854,Z 695.985,A -85,B 0,C 180,E1 -15117.565,E2 -15117.565} C_VEL
LIN {X 0,Y 332.142,Z 684.689,A -85,B 0,C 180,E1 -15118.787,E2 -15118.787} C_VEL
LIN {X 0,Y 333.219,Z 672.032,A -85,B 0,C 180,E1 -15119.849,E2 -15119.849} C_VEL
LIN {X 0,Y 333.885,Z 659.295,A -85,B 0,C 180,E1 -15120.641,E2 -15120.641} C_VEL
LIN {X 0,Y 334.194,Z 646.212,A -85,B 0,C 180,E1 -15121.205,E2 -15121.205} C_VEL
LIN {X 0,Y 335.091,Z 616.708,A -85,B 0,C 180,E1 -15122.105,E2 -15122.105} C_VEL
LIN {X 0,Y 336.239,Z 590.712,A -85,B 0,C 180,E1 -15122.881,E2 -15122.881} C_VEL
LIN {X 0,Y 332.552,Z 583.107,A -85,B 0,C 180,E1 -15123.62,E2 -15123.62} C_VEL
LIN {X 0,Y 328.408,Z 575.625,A -85,B 0,C 180,E1 -15124.459,E2 -15124.459} C_VEL
LIN {X 0,Y 323.665,Z 567.956,A -85,B 0,C 180,E1 -15125.447,E2 -15125.447} C_VEL
LIN {X 0,Y 321.701,Z 564.555,A -85,B 0,C 180,E1 -15125.883,E2 -15125.883} C_VEL
LIN {X 0,Y 320.19,Z 561.813,A -85,B 0,C 180,E1 -15126.242,E2 -15126.242} C_VEL
LIN {X 0,Y 319.954,Z 560.633,A -85,B 0,C 180,E1 -15126.385,E2 -15126.385} C_VEL
LIN {X 0,Y 319.833,Z 560.647,A -85,B 0,C 180,E1 -15128.848,E2 -15128.848} C_VEL
LIN {X 0,Y 319.675,Z 560.659,A -85,B 0,C 180,E1 -15132.7,E2 -15132.7} C_VEL
LIN {X 0,Y 319.69,Z 560.656,A -85,B 0,C 180,E1 -15135.296,E2 -15135.296} C_VEL
LIN {X 0,Y 319.665,Z 560.666,A -85,B 0,C 180,E1 -15139.256,E2 -15139.256} C_VEL
LIN {X 0,Y 319.561,Z 560.679,A -85,B 0,C 180,E1 -15143.32,E2 -15143.32} C_VEL
LIN {X 0,Y 319.626,Z 560.669,A -85,B 0,C 180,E1 -15146.089,E2 -15146.089} C_VEL
LIN {X 0,Y 319.581,Z 560.676,A -85,B 0,C 180,E1 -15148.934,E2 -15148.934} C_VEL
LIN {X 0,Y 319.524,Z 560.684,A -85,B 0,C 180,E1 -15151.863,E2 -15151.863} C_VEL
LIN {X 0,Y 319.573,Z 560.675,A -85,B 0,C 180,E1 -15155.544,E2 -15155.544} C_VEL
LIN {X 0,Y 319.593,Z 560.67,A -85,B 0,C 180,E1 -15158.005,E2 -15158.005} C_VEL
LIN {X 0,Y 319.595,Z 560.678,A -85,B 0,C 180,E1 -15161.614,E2 -15161.614} C_VEL
LIN {X 0,Y 319.64,Z 560.668,A -85,B 0,C 180,E1 -15165.287,E2 -15165.287} C_VEL
LIN {X 0,Y 319.597,Z 560.712,A -85,B 0,C 180,E1 -15167.118,E2 -15167.118} C_VEL
LIN {X 0,Y 322.554,Z 570.094,A -85,B 0,C 180,E1 -15170.814,E2 -15170.814} C_VEL
LIN {X 0,Y 325.21,Z 579.534,A -85,B 0,C 180,E1 -15173.991,E2 -15173.991} C_VEL
LIN {X 0,Y 327.374,Z 589.271,A -85,B 0,C 180,E1 -15176.85,E2 -15176.85} C_VEL
LIN {X 0,Y 328.451,Z 595.01,A -85,B 0,C 180,E1 -15178.386,E2 -15178.386} C_VEL
LIN {X 0,Y 328.285,Z 597.967,A -85,B 0,C 180,E1 -15179.085,E2 -15179.085} C_VEL
LIN {X 0,Y 325.843,Z 612.349,A -85,B 0,C 180,E1 -15182.168,E2 -15182.168} C_VEL
LIN {X 0,Y 329.47,Z 633.649,A -85,B 0,C 180,E1 -15183.41,E2 -15183.41} C_VEL
LIN {X 0,Y 331.684,Z 651.765,A -85,B 0,C 180,E1 -15184.298,E2 -15184.298} C_VEL
LIN {X 0,Y 333.115,Z 672.449,A -85,B 0,C 180,E1 -15185.157,E2 -15185.157} C_VEL
LIN {X 0,Y 333.344,Z 681.287,A -85,B 0,C 180,E1 -15185.479,E2 -15185.479} C_VEL
LIN {X 0,Y 331.297,Z 727.826,A -85,B 0,C 180,E1 -15186.812,E2 -15186.812} C_VEL
LIN {X 0,Y 330.157,Z 740.988,A -85,B 0,C 180,E1 -15187.389,E2 -15187.389} C_VEL
LIN {X 0,Y 328.6,Z 753.93,A -85,B 0,C 180,E1 -15188.186,E2 -15188.186} C_VEL
LIN {X 0,Y 327.475,Z 770.523,A -85,B 0,C 180,E1 -15188.934,E2 -15188.934} C_VEL
LIN {X 0,Y 326.444,Z 782.142,A -85,B 0,C 180,E1 -15189.688,E2 -15189.688} C_VEL
LIN {X 0,Y 325.171,Z 794.388,A -85,B 0,C 180,E1 -15190.757,E2 -15190.757} C_VEL
LIN {X 0,Y 323.845,Z 805.306,A -85,B 0,C 180,E1 -15191.987,E2 -15191.987} C_VEL
LIN {X 0,Y 322.686,Z 814.155,A -85,B 0,C 180,E1 -15193.228,E2 -15193.228} C_VEL
LIN {X 0,Y 321.424,Z 823.241,A -85,B 0,C 180,E1 -15194.79,E2 -15194.79} C_VEL
LIN {X 0,Y 320.213,Z 832.086,A -85,B 0,C 180,E1 -15196.678,E2 -15196.678} C_VEL
LIN {X 0,Y 319.208,Z 839.161,A -85,B 0,C 180,E1 -15198.572,E2 -15198.572} C_VEL
LIN {X 0,Y 318.591,Z 844.786,A -85,B 0,C 180,E1 -15200.478,E2 -15200.478} C_VEL
LIN {X 0,Y 318.142,Z 849.197,A -85,B 0,C 180,E1 -15202.385,E2 -15202.385} C_VEL
LIN {X 0,Y 317.935,Z 852.272,A -85,B 0,C 180,E1 -15204.117,E2 -15204.117} C_VEL
LIN {X 0,Y 317.902,Z 854.843,A -85,B 0,C 180,E1 -15206.198,E2 -15206.198} C_VEL
LIN {X 0,Y 317.855,Z 856.465,A -85,B 0,C 180,E1 -15208.734,E2 -15208.734} C_VEL
LIN {X 0,Y 317.917,Z 856.684,A -85,B 0,C 180,E1 -15210.001,E2 -15210.001} C_VEL
LIN {X 0,Y 317.842,Z 855.837,A -85,B 0,C 180,E1 -15212.536,E2 -15212.536} C_VEL
LIN {X 0,Y 317.894,Z 854.826,A -85,B 0,C 180,E1 -15213.804,E2 -15213.804} C_VEL
LIN {X 0,Y 317.923,Z 852.277,A -85,B 0,C 180,E1 -15215.862,E2 -15215.862} C_VEL
LIN {X 0,Y 318.175,Z 849.161,A -85,B 0,C 180,E1 -15217.617,E2 -15217.617} C_VEL
LIN {X 0,Y 318.577,Z 844.739,A -85,B 0,C 180,E1 -15219.525,E2 -15219.525} C_VEL
LIN {X 0,Y 319.304,Z 837.999,A -85,B 0,C 180,E1 -15221.748,E2 -15221.748} C_VEL
LIN {X 0,Y 320.362,Z 830.648,A -85,B 0,C 180,E1 -15223.641,E2 -15223.641} C_VEL
LIN {X 0,Y 321.597,Z 821.888,A -85,B 0,C 180,E1 -15225.454,E2 -15225.454} C_VEL
LIN {X 0,Y 322.864,Z 811.936,A -85,B 0,C 180,E1 -15227.09,E2 -15227.09} C_VEL
LIN {X 0,Y 324.285,Z 801.333,A -85,B 0,C 180,E1 -15228.48,E2 -15228.48} C_VEL
LIN {X 0,Y 325.54,Z 791.058,A -85,B 0,C 180,E1 -15229.551,E2 -15229.551} C_VEL
LIN {X 0,Y 326.715,Z 778.708,A -85,B 0,C 180,E1 -15230.543,E2 -15230.543} C_VEL
LIN {X 0,Y 327.766,Z 765.72,A -85,B 0,C 180,E1 -15231.296,E2 -15231.296} C_VEL
LIN {X 0,Y 328.517,Z 752.646,A -85,B 0,C 180,E1 -15231.78,E2 -15231.78} C_VEL
LIN {X 0,Y 330.005,Z 679.452,A -85,B 0,C 180,E1 -15233.381,E2 -15233.381} C_VEL
LIN {X 0,Y 326.632,Z 648.324,A -85,B 0,C 180,E1 -15234.366,E2 -15234.366} C_VEL
LIN {X 0,Y 324.863,Z 635.633,A -85,B 0,C 180,E1 -15234.819,E2 -15234.819} C_VEL
LIN {X 0,Y 323.286,Z 614.436,A -85,B 0,C 180,E1 -15236.425,E2 -15236.425} C_VEL
LIN {X 0,Y 323.098,Z 611.214,A -85,B 0,C 180,E1 -15236.67,E2 -15236.67} C_VEL
LIN {X 0,Y 325.527,Z 590.837,A -85,B 0,C 180,E1 -15241.209,E2 -15241.209} C_VEL
LIN {X 0,Y 325.472,Z 587.694,A -85,B 0,C 180,E1 -15241.941,E2 -15241.941} C_VEL
LIN {X 0,Y 322.637,Z 574.308,A -85,B 0,C 180,E1 -15245.258,E2 -15245.258} C_VEL
LIN {X 0,Y 319.604,Z 560.675,A -85,B 0,C 180,E1 -15248.859,E2 -15248.859} C_VEL
LIN {X 0,Y 319.562,Z 560.674,A -85,B 0,C 180,E1 -15252.983,E2 -15252.983} C_VEL
LIN {X 0,Y 319.564,Z 560.675,A -85,B 0,C 180,E1 -15257.018,E2 -15257.018} C_VEL
LIN {X 0,Y 319.549,Z 560.679,A -85,B 0,C 180,E1 -15260.371,E2 -15260.371} C_VEL
LIN {X 0,Y 319.582,Z 560.668,A -85,B 0,C 180,E1 -15264.457,E2 -15264.457} C_VEL
LIN {X 0,Y 319.534,Z 560.67,A -85,B 0,C 180,E1 -15268.138,E2 -15268.138} C_VEL
LIN {X 0,Y 319.618,Z 560.674,A -85,B 0,C 180,E1 -15271.589,E2 -15271.589} C_VEL
LIN {X 0,Y 319.604,Z 560.654,A -85,B 0,C 180,E1 -15275.304,E2 -15275.304} C_VEL
LIN {X 0,Y 319.603,Z 560.672,A -85,B 0,C 180,E1 -15279.4,E2 -15279.4} C_VEL
LIN {X 0,Y 319.659,Z 560.642,A -85,B 0,C 180,E1 -15282.073,E2 -15282.073} C_VEL
LIN {X 0,Y 319.733,Z 560.656,A -85,B 0,C 180,E1 -15286.008,E2 -15286.008} C_VEL
LIN {X 0,Y 319.753,Z 560.631,A -85,B 0,C 180,E1 -15289.873,E2 -15289.873} C_VEL
LIN {X 0,Y 319.914,Z 560.632,A -85,B 0,C 180,E1 -15292.426,E2 -15292.426} C_VEL
LIN {X 0,Y 319.747,Z 560.653,A -85,B 0,C 180,E1 -15294.956,E2 -15294.956} C_VEL
LIN {X 0,Y 319.99,Z 560.6,A -85,B 0,C 180,E1 -15297.482,E2 -15297.482} C_VEL
LIN {X 0,Y 320.132,Z 560.605,A -85,B 0,C 180,E1 -15300,E2 -15300} C_VEL
LIN {X 0,Y 319.991,Z 560.62,A -85,B 0,C 180,E1 -15302.518,E2 -15302.518} C_VEL
LIN {X 0,Y 319.927,Z 560.618,A -85,B 0,C 180,E1 -15306.628,E2 -15306.628} C_VEL
LIN {X 0,Y 319.844,Z 560.642,A -85,B 0,C 180,E1 -15308.848,E2 -15308.848} C_VEL
LIN {X 0,Y 319.682,Z 560.641,A -85,B 0,C 180,E1 -15312.7,E2 -15312.7} C_VEL
LIN {X 0,Y 319.701,Z 560.659,A -85,B 0,C 180,E1 -15315.296,E2 -15315.296} C_VEL
LIN {X 0,Y 319.676,Z 560.644,A -85,B 0,C 180,E1 -15319.255,E2 -15319.255} C_VEL
LIN {X 0,Y 319.572,Z 560.677,A -85,B 0,C 180,E1 -15323.319,E2 -15323.319} C_VEL
LIN {X 0,Y 319.62,Z 560.658,A -85,B 0,C 180,E1 -15326.09,E2 -15326.09} C_VEL
LIN {X 0,Y 319.582,Z 560.674,A -85,B 0,C 180,E1 -15328.935,E2 -15328.935} C_VEL
LIN {X 0,Y 319.534,Z 560.675,A -85,B 0,C 180,E1 -15331.862,E2 -15331.862} C_VEL
LIN {X 0,Y 319.582,Z 560.667,A -85,B 0,C 180,E1 -15335.543,E2 -15335.543} C_VEL
LIN {X 0,Y 319.575,Z 560.682,A -85,B 0,C 180,E1 -15338.008,E2 -15338.008} C_VEL
LIN {X 0,Y 319.528,Z 560.686,A -85,B 0,C 180,E1 -15341.597,E2 -15341.597} C_VEL
LIN {X 0,Y 319.49,Z 560.687,A -85,B 0,C 180,E1 -15345.257,E2 -15345.257} C_VEL
LIN {X 0,Y 319.53,Z 560.668,A -85,B 0,C 180,E1 -15348.711,E2 -15348.711} C_VEL
LIN {X 0,Y 319.579,Z 560.695,A -85,B 0,C 180,E1 -15352.617,E2 -15352.617} C_VEL
LIN {X 0,Y 323.505,Z 573.88,A -85,B 0,C 180,E1 -15355.643,E2 -15355.643} C_VEL
LIN {X 0,Y 326.839,Z 587.278,A -85,B 0,C 180,E1 -15358.576,E2 -15358.576} C_VEL
LIN {X 0,Y 328.723,Z 596.826,A -85,B 0,C 180,E1 -15360.545,E2 -15360.545} C_VEL
LIN {X 0,Y 327.077,Z 616.102,A -85,B 0,C 180,E1 -15363.864,E2 -15363.864} C_VEL
LIN {X 0,Y 326.595,Z 624.481,A -85,B 0,C 180,E1 -15365.248,E2 -15365.248} C_VEL
LIN {X 0,Y 331.123,Z 653.234,A -85,B 0,C 180,E1 -15366.285,E2 -15366.285} C_VEL
LIN {X 0,Y 329.265,Z 736.034,A -85,B 0,C 180,E1 -15368.107,E2 -15368.107} C_VEL
LIN {X 0,Y 328.579,Z 749.465,A -85,B 0,C 180,E1 -15368.636,E2 -15368.636} C_VEL
LIN {X 0,Y 327.556,Z 762.554,A -85,B 0,C 180,E1 -15369.43,E2 -15369.43} C_VEL
LIN {X 0,Y 326.505,Z 773.701,A -85,B 0,C 180,E1 -15370.346,E2 -15370.346} C_VEL
LIN {X 0,Y 325.27,Z 783.972,A -85,B 0,C 180,E1 -15371.415,E2 -15371.415} C_VEL
LIN {X 0,Y 324.068,Z 794.422,A -85,B 0,C 180,E1 -15372.798,E2 -15372.798} C_VEL
LIN {X 0,Y 322.835,Z 803.138,A -85,B 0,C 180,E1 -15374.209,E2 -15374.209} C_VEL
LIN {X 0,Y 321.364,Z 812.508,A -85,B 0,C 180,E1 -15376.079,E2 -15376.079} C_VEL
LIN {X 0,Y 320.238,Z 819.954,A -85,B 0,C 180,E1 -15377.965,E2 -15377.965} C_VEL
LIN {X 0,Y 319.371,Z 825.933,A -85,B 0,C 180,E1 -15379.86,E2 -15379.86} C_VEL
LIN {X 0,Y 318.72,Z 830.659,A -85,B 0,C 180,E1 -15381.759,E2 -15381.759} C_VEL
LIN {X 0,Y 318.316,Z 834.271,A -85,B 0,C 180,E1 -15383.661,E2 -15383.661} C_VEL
LIN {X 0,Y 318.124,Z 836.13,A -85,B 0,C 180,E1 -15384.929,E2 -15384.929} C_VEL
LIN {X 0,Y 317.978,Z 837.55,A -85,B 0,C 180,E1 -15386.197,E2 -15386.197} C_VEL
LIN {X 0,Y 317.782,Z 839.161,A -85,B 0,C 180,E1 -15388.732,E2 -15388.732} C_VEL
LIN {X 0,Y 317.786,Z 839.394,A -85,B 0,C 180,E1 -15389.999,E2 -15389.999} C_VEL
LIN {X 0,Y 317.781,Z 839.201,A -85,B 0,C 180,E1 -15391.266,E2 -15391.266} C_VEL
LIN {X 0,Y 317.972,Z 837.646,A -85,B 0,C 180,E1 -15393.801,E2 -15393.801} C_VEL
LIN {X 0,Y 318.12,Z 836.278,A -85,B 0,C 180,E1 -15395.069,E2 -15395.069} C_VEL
LIN {X 0,Y 318.342,Z 834.095,A -85,B 0,C 180,E1 -15396.554,E2 -15396.554} C_VEL
LIN {X 0,Y 318.882,Z 829.497,A -85,B 0,C 180,E1 -15398.874,E2 -15398.874} C_VEL
LIN {X 0,Y 319.609,Z 824.435,A -85,B 0,C 180,E1 -15400.771,E2 -15400.771} C_VEL
LIN {X 0,Y 320.542,Z 818.054,A -85,B 0,C 180,E1 -15402.664,E2 -15402.664} C_VEL
LIN {X 0,Y 321.767,Z 810.11,A -85,B 0,C 180,E1 -15404.546,E2 -15404.546} C_VEL
LIN {X 0,Y 323.078,Z 801.982,A -85,B 0,C 180,E1 -15406.101,E2 -15406.101} C_VEL
LIN {X 0,Y 324.349,Z 792.001,A -85,B 0,C 180,E1 -15407.658,E2 -15407.658} C_VEL
LIN {X 0,Y 325.724,Z 780.778,A -85,B 0,C 180,E1 -15409.046,E2 -15409.046} C_VEL
LIN {X 0,Y 326.958,Z 769.748,A -85,B 0,C 180,E1 -15410.115,E2 -15410.115} C_VEL
LIN {X 0,Y 328.125,Z 757.281,A -85,B 0,C 180,E1 -15411.023,E2 -15411.023} C_VEL
LIN {X 0,Y 328.838,Z 745.086,A -85,B 0,C 180,E1 -15411.673,E2 -15411.673} C_VEL
LIN {X 0,Y 329.393,Z 733,A -85,B 0,C 180,E1 -15412.088,E2 -15412.088} C_VEL
LIN {X 0,Y 331.022,Z 655.06,A -85,B 0,C 180,E1 -15413.789,E2 -15413.789} C_VEL
LIN {X 0,Y 327.031,Z 631.549,A -85,B 0,C 180,E1 -15414.656,E2 -15414.656} C_VEL
LIN {X 0,Y 325.803,Z 625.076,A -85,B 0,C 180,E1 -15414.948,E2 -15414.948} C_VEL
LIN {X 0,Y 327.137,Z 607.431,A -85,B 0,C 180,E1 -15418.258,E2 -15418.258} C_VEL
LIN {X 0,Y 327.243,Z 605.972,A -85,B 0,C 180,E1 -15418.537,E2 -15418.537} C_VEL
LIN {X 0,Y 326.943,Z 602.271,A -85,B 0,C 180,E1 -15419.335,E2 -15419.335} C_VEL
LIN {X 0,Y 325.563,Z 598.906,A -85,B 0,C 180,E1 -15420.164,E2 -15420.164} C_VEL
LIN {X 0,Y 320.443,Z 590.577,A -85,B 0,C 180,E1 -15422.453,E2 -15422.453} C_VEL
LIN {X 0,Y 319.633,Z 588.278,A -85,B 0,C 180,E1 -15423.033,E2 -15423.033} C_VEL
LIN {X 0,Y 316.745,Z 576.343,A -85,B 0,C 180,E1 -15425.954,E2 -15425.954} C_VEL
LIN {X 0,Y 313.542,Z 565.109,A -85,B 0,C 180,E1 -15428.872,E2 -15428.872} C_VEL
LIN {X 0,Y 312.514,Z 561.547,A -85,B 0,C 180,E1 -15429.848,E2 -15429.848} C_VEL
LIN {X 0,Y 312.507,Z 561.539,A -85,B 0,C 180,E1 -15434.197,E2 -15434.197} C_VEL
LIN {X 0,Y 312.549,Z 561.586,A -85,B 0,C 180,E1 -15435.038,E2 -15435.038} C_VEL
LIN {X 0,Y 320.661,Z 584.403,A -85,B 0,C 180,E1 -15436.159,E2 -15436.159} C_VEL
LIN {X 0,Y 319.459,Z 636.344,A -85,B 0,C 180,E1 -15437.578,E2 -15437.578} C_VEL
LIN {X 0,Y 319.303,Z 650.4,A -85,B 0,C 180,E1 -15438.103,E2 -15438.103} C_VEL
LIN {X 0,Y 318.935,Z 663.289,A -85,B 0,C 180,E1 -15438.828,E2 -15438.828} C_VEL
LIN {X 0,Y 318.313,Z 675.631,A -85,B 0,C 180,E1 -15439.773,E2 -15439.773} C_VEL
LIN {X 0,Y 317.551,Z 688.218,A -85,B 0,C 180,E1 -15441.03,E2 -15441.03} C_VEL
LIN {X 0,Y 316.691,Z 699.581,A -85,B 0,C 180,E1 -15442.47,E2 -15442.47} C_VEL
LIN {X 0,Y 315.847,Z 709.703,A -85,B 0,C 180,E1 -15444.064,E2 -15444.064} C_VEL
LIN {X 0,Y 315.036,Z 718.382,A -85,B 0,C 180,E1 -15445.73,E2 -15445.73} C_VEL
LIN {X 0,Y 314.347,Z 726.079,A -85,B 0,C 180,E1 -15447.549,E2 -15447.549} C_VEL
LIN {X 0,Y 313.649,Z 733.442,A -85,B 0,C 180,E1 -15449.724,E2 -15449.724} C_VEL
LIN {X 0,Y 313.254,Z 739.114,A -85,B 0,C 180,E1 -15451.891,E2 -15451.891} C_VEL
LIN {X 0,Y 312.974,Z 743.097,A -85,B 0,C 180,E1 -15453.921,E2 -15453.921} C_VEL
LIN {X 0,Y 312.837,Z 746.164,A -85,B 0,C 180,E1 -15456.148,E2 -15456.148} C_VEL
LIN {X 0,Y 312.909,Z 747.462,A -85,B 0,C 180,E1 -15457.553,E2 -15457.553} C_VEL
LIN {X 0,Y 313.035,Z 748.212,A -85,B 0,C 180,E1 -15458.948,E2 -15458.948} C_VEL
LIN {X 0,Y 313.281,Z 748.5,A -85,B 0,C 180,E1 -15460.42,E2 -15460.42} C_VEL
LIN {X 0,Y 313.569,Z 748.302,A -85,B 0,C 180,E1 -15461.713,E2 -15461.713} C_VEL
LIN {X 0,Y 314.306,Z 746.832,A -85,B 0,C 180,E1 -15464.042,E2 -15464.042} C_VEL
LIN {X 0,Y 315.352,Z 743.814,A -85,B 0,C 180,E1 -15466.467,E2 -15466.467} C_VEL
LIN {X 0,Y 316.402,Z 740.03,A -85,B 0,C 180,E1 -15468.468,E2 -15468.468} C_VEL
LIN {X 0,Y 317.711,Z 734.956,A -85,B 0,C 180,E1 -15470.45,E2 -15470.45} C_VEL
LIN {X 0,Y 319.156,Z 728.502,A -85,B 0,C 180,E1 -15472.408,E2 -15472.408} C_VEL
LIN {X 0,Y 320.829,Z 720.437,A -85,B 0,C 180,E1 -15474.343,E2 -15474.343} C_VEL
LIN {X 0,Y 322.392,Z 712.06,A -85,B 0,C 180,E1 -15475.937,E2 -15475.937} C_VEL
LIN {X 0,Y 323.948,Z 701.874,A -85,B 0,C 180,E1 -15477.513,E2 -15477.513} C_VEL
LIN {X 0,Y 325.339,Z 691.73,A -85,B 0,C 180,E1 -15478.762,E2 -15478.762} C_VEL
LIN {X 0,Y 326.492,Z 680.693,A -85,B 0,C 180,E1 -15479.846,E2 -15479.846} C_VEL
LIN {X 0,Y 327.572,Z 667.443,A -85,B 0,C 180,E1 -15480.845,E2 -15480.845} C_VEL
LIN {X 0,Y 328.074,Z 654.99,A -85,B 0,C 180,E1 -15481.534,E2 -15481.534} C_VEL
LIN {X 0,Y 328.448,Z 637.055,A -85,B 0,C 180,E1 -15482.184,E2 -15482.184} C_VEL
LIN {X 0,Y 330.434,Z 593.106,A -85,B 0,C 180,E1 -15483.523,E2 -15483.523} C_VEL
LIN {X 0,Y 324.975,Z 582.284,A -85,B 0,C 180,E1 -15484.684,E2 -15484.684} C_VEL
LIN {X 0,Y 316.584,Z 568.332,A -85,B 0,C 180,E1 -15486.553,E2 -15486.553} C_VEL
LIN {X 0,Y 315.126,Z 565.847,A -85,B 0,C 180,E1 -15486.905,E2 -15486.905} C_VEL
LIN {X 0,Y 313.398,Z 563.4,A -85,B 0,C 180,E1 -15487.307,E2 -15487.307} C_VEL
LIN {X 0,Y 312.9,Z 561.503,A -85,B 0,C 180,E1 -15487.502,E2 -15487.502} C_VEL
LIN {X 0,Y 312.662,Z 561.539,A -85,B 0,C 180,E1 -15491.672,E2 -15491.672} C_VEL
LIN {X 0,Y 312.69,Z 561.531,A -85,B 0,C 180,E1 -15494.888,E2 -15494.888} C_VEL
LIN {X 0,Y 312.621,Z 561.543,A -85,B 0,C 180,E1 -15499.237,E2 -15499.237} C_VEL
LIN {X 0,Y 312.537,Z 561.553,A -85,B 0,C 180,E1 -15502.79,E2 -15502.79} C_VEL
LIN {X 0,Y 312.594,Z 561.545,A -85,B 0,C 180,E1 -15505.936,E2 -15505.936} C_VEL
LIN {X 0,Y 312.537,Z 561.553,A -85,B 0,C 180,E1 -15509.651,E2 -15509.651} C_VEL
LIN {X 0,Y 312.511,Z 561.556,A -85,B 0,C 180,E1 -15513.69,E2 -15513.69} C_VEL
LIN {X 0,Y 312.534,Z 561.548,A -85,B 0,C 180,E1 -15517.384,E2 -15517.384} C_VEL
LIN {X 0,Y 312.529,Z 561.552,A -85,B 0,C 180,E1 -15520.703,E2 -15520.703} C_VEL
LIN {X 0,Y 312.589,Z 561.551,A -85,B 0,C 180,E1 -15524.185,E2 -15524.185} C_VEL
LIN {X 0,Y 312.589,Z 561.603,A -85,B 0,C 180,E1 -15525.817,E2 -15525.817} C_VEL
LIN {X 0,Y 315.143,Z 569.681,A -85,B 0,C 180,E1 -15529.309,E2 -15529.309} C_VEL
LIN {X 0,Y 317.549,Z 577.936,A -85,B 0,C 180,E1 -15532.362,E2 -15532.362} C_VEL
LIN {X 0,Y 319.726,Z 586.569,A -85,B 0,C 180,E1 -15535.146,E2 -15535.146} C_VEL
LIN {X 0,Y 321.687,Z 596.551,A -85,B 0,C 180,E1 -15538.01,E2 -15538.01} C_VEL
LIN {X 0,Y 321.693,Z 599.173,A -85,B 0,C 180,E1 -15538.662,E2 -15538.662} C_VEL
LIN {X 0,Y 319.569,Z 610.749,A -85,B 0,C 180,E1 -15541.227,E2 -15541.227} C_VEL
LIN {X 0,Y 323.225,Z 631.832,A -85,B 0,C 180,E1 -15542.544,E2 -15542.544} C_VEL
LIN {X 0,Y 325.694,Z 651.904,A -85,B 0,C 180,E1 -15543.595,E2 -15543.595} C_VEL
LIN {X 0,Y 327.084,Z 672.22,A -85,B 0,C 180,E1 -15544.482,E2 -15544.482} C_VEL
LIN {X 0,Y 327.269,Z 682.656,A -85,B 0,C 180,E1 -15544.861,E2 -15544.861} C_VEL
LIN {X 0,Y 325.211,Z 726.327,A -85,B 0,C 180,E1 -15546.14,E2 -15546.14} C_VEL
LIN {X 0,Y 323.946,Z 740.101,A -85,B 0,C 180,E1 -15546.762,E2 -15546.762} C_VEL
LIN {X 0,Y 322.364,Z 752.817,A -85,B 0,C 180,E1 -15547.573,E2 -15547.573} C_VEL
LIN {X 0,Y 321.739,Z 756.722,A -85,B 0,C 180,E1 -15547.866,E2 -15547.866} C_VEL
LIN {X 0,Y 320.983,Z 768.923,A -85,B 0,C 180,E1 -15548.402,E2 -15548.402} C_VEL
LIN {X 0,Y 319.922,Z 780.995,A -85,B 0,C 180,E1 -15549.171,E2 -15549.171} C_VEL
LIN {X 0,Y 318.649,Z 792.649,A -85,B 0,C 180,E1 -15550.179,E2 -15550.179} C_VEL
LIN {X 0,Y 317.232,Z 803.87,A -85,B 0,C 180,E1 -15551.431,E2 -15551.431} C_VEL
LIN {X 0,Y 315.868,Z 813.972,A -85,B 0,C 180,E1 -15552.855,E2 -15552.855} C_VEL
LIN {X 0,Y 314.563,Z 823.055,A -85,B 0,C 180,E1 -15554.45,E2 -15554.45} C_VEL
LIN {X 0,Y 313.259,Z 831.898,A -85,B 0,C 180,E1 -15556.376,E2 -15556.376} C_VEL
LIN {X 0,Y 312.201,Z 838.971,A -85,B 0,C 180,E1 -15558.312,E2 -15558.312} C_VEL
LIN {X 0,Y 311.543,Z 844.595,A -85,B 0,C 180,E1 -15560.261,E2 -15560.261} C_VEL
LIN {X 0,Y 311.068,Z 849.004,A -85,B 0,C 180,E1 -15562.21,E2 -15562.21} C_VEL
LIN {X 0,Y 310.848,Z 852.32,A -85,B 0,C 180,E1 -15564.158,E2 -15564.158} C_VEL
LIN {X 0,Y 310.81,Z 854.65,A -85,B 0,C 180,E1 -15566.111,E2 -15566.111} C_VEL
LIN {X 0,Y 310.768,Z 855.657,A -85,B 0,C 180,E1 -15567.409,E2 -15567.409} C_VEL
LIN {X 0,Y 310.763,Z 856.272,A -85,B 0,C 180,E1 -15568.705,E2 -15568.705} C_VEL
LIN {X 0,Y 310.821,Z 856.491,A -85,B 0,C 180,E1 -15570.001,E2 -15570.001} C_VEL
LIN {X 0,Y 310.763,Z 855.644,A -85,B 0,C 180,E1 -15572.593,E2 -15572.593} C_VEL
LIN {X 0,Y 310.801,Z 854.632,A -85,B 0,C 180,E1 -15573.891,E2 -15573.891} C_VEL
LIN {X 0,Y 310.848,Z 852.293,A -85,B 0,C 180,E1 -15575.844,E2 -15575.844} C_VEL
LIN {X 0,Y 311.098,Z 848.967,A -85,B 0,C 180,E1 -15577.791,E2 -15577.791} C_VEL
LIN {X 0,Y 311.53,Z 844.545,A -85,B 0,C 180,E1 -15579.742,E2 -15579.742} C_VEL
LIN {X 0,Y 312.172,Z 838.902,A -85,B 0,C 180,E1 -15581.691,E2 -15581.691} C_VEL
LIN {X 0,Y 313.228,Z 831.806,A -85,B 0,C 180,E1 -15583.627,E2 -15583.627} C_VEL
LIN {X 0,Y 314.535,Z 822.957,A -85,B 0,C 180,E1 -15585.554,E2 -15585.554} C_VEL
LIN {X 0,Y 315.91,Z 812.811,A -85,B 0,C 180,E1 -15587.311,E2 -15587.311} C_VEL
LIN {X 0,Y 317.364,Z 802.429,A -85,B 0,C 180,E1 -15588.73,E2 -15588.73} C_VEL
LIN {X 0,Y 318.843,Z 790.877,A -85,B 0,C 180,E1 -15589.978,E2 -15589.978} C_VEL
LIN {X 0,Y 320.071,Z 778.535,A -85,B 0,C 180,E1 -15590.989,E2 -15590.989} C_VEL
LIN {X 0,Y 321.168,Z 765.56,A -85,B 0,C 180,E1 -15591.756,E2 -15591.756} C_VEL
LIN {X 0,Y 321.948,Z 752.525,A -85,B 0,C 180,E1 -15592.248,E2 -15592.248} C_VEL
LIN {X 0,Y 323.518,Z 680.402,A -85,B 0,C 180,E1 -15593.854,E2 -15593.854} C_VEL
LIN {X 0,Y 320.172,Z 649.272,A -85,B 0,C 180,E1 -15594.866,E2 -15594.866} C_VEL
LIN {X 0,Y 318.285,Z 635.467,A -85,B 0,C 180,E1 -15595.376,E2 -15595.376} C_VEL
LIN {X 0,Y 316.744,Z 613.629,A -85,B 0,C 180,E1 -15597.089,E2 -15597.089} C_VEL
LIN {X 0,Y 316.36,Z 608.922,A -85,B 0,C 180,E1 -15597.466,E2 -15597.466} C_VEL
LIN {X 0,Y 318.471,Z 592.321,A -85,B 0,C 180,E1 -15601.239,E2 -15601.239} C_VEL
LIN {X 0,Y 318.535,Z 589.183,A -85,B 0,C 180,E1 -15601.974,E2 -15601.974} C_VEL
LIN {X 0,Y 315.712,Z 575.831,A -85,B 0,C 180,E1 -15605.365,E2 -15605.365} C_VEL
LIN {X 0,Y 312.567,Z 561.552,A -85,B 0,C 180,E1 -15609.169,E2 -15609.169} C_VEL
LIN {X 0,Y 312.495,Z 561.56,A -85,B 0,C 180,E1 -15612.431,E2 -15612.431} C_VEL
LIN {X 0,Y 312.484,Z 561.56,A -85,B 0,C 180,E1 -15616.031,E2 -15616.031} C_VEL
LIN {X 0,Y 312.506,Z 561.557,A -85,B 0,C 180,E1 -15619.875,E2 -15619.875} C_VEL
LIN {X 0,Y 312.537,Z 561.542,A -85,B 0,C 180,E1 -15624.05,E2 -15624.05} C_VEL
LIN {X 0,Y 312.506,Z 561.551,A -85,B 0,C 180,E1 -15627.334,E2 -15627.334} C_VEL
LIN {X 0,Y 312.554,Z 561.55,A -85,B 0,C 180,E1 -15631.276,E2 -15631.276} C_VEL
LIN {X 0,Y 312.586,Z 561.53,A -85,B 0,C 180,E1 -15634.711,E2 -15634.711} C_VEL
LIN {X 0,Y 312.539,Z 561.554,A -85,B 0,C 180,E1 -15638.913,E2 -15638.913} C_VEL
LIN {X 0,Y 312.639,Z 561.518,A -85,B 0,C 180,E1 -15641.656,E2 -15641.656} C_VEL
LIN {X 0,Y 312.695,Z 561.536,A -85,B 0,C 180,E1 -15645.686,E2 -15645.686} C_VEL
LIN {X 0,Y 312.699,Z 561.509,A -85,B 0,C 180,E1 -15649.642,E2 -15649.642} C_VEL
LIN {X 0,Y 312.855,Z 561.512,A -85,B 0,C 180,E1 -15652.254,E2 -15652.254} C_VEL
LIN {X 0,Y 312.717,Z 561.528,A -85,B 0,C 180,E1 -15654.842,E2 -15654.842} C_VEL
LIN {X 0,Y 312.989,Z 561.483,A -85,B 0,C 180,E1 -15658.713,E2 -15658.713} C_VEL
LIN {X 0,Y 312.991,Z 561.498,A -85,B 0,C 180,E1 -15661.287,E2 -15661.287} C_VEL
LIN {X 0,Y 312.717,Z 561.505,A -85,B 0,C 180,E1 -15665.158,E2 -15665.158} C_VEL
LIN {X 0,Y 312.868,Z 561.509,A -85,B 0,C 180,E1 -15667.746,E2 -15667.746} C_VEL
LIN {X 0,Y 312.671,Z 561.517,A -85,B 0,C 180,E1 -15671.671,E2 -15671.671} C_VEL
LIN {X 0,Y 312.702,Z 561.53,A -85,B 0,C 180,E1 -15674.888,E2 -15674.888} C_VEL
LIN {X 0,Y 312.632,Z 561.521,A -85,B 0,C 180,E1 -15679.236,E2 -15679.236} C_VEL
LIN {X 0,Y 312.548,Z 561.551,A -85,B 0,C 180,E1 -15682.789,E2 -15682.789} C_VEL
LIN {X 0,Y 312.599,Z 561.531,A -85,B 0,C 180,E1 -15685.933,E2 -15685.933} C_VEL
LIN {X 0,Y 312.54,Z 561.547,A -85,B 0,C 180,E1 -15689.651,E2 -15689.651} C_VEL
LIN {X 0,Y 312.522,Z 561.559,A -85,B 0,C 180,E1 -15693.689,E2 -15693.689} C_VEL
LIN {X 0,Y 312.539,Z 561.556,A -85,B 0,C 180,E1 -15697.383,E2 -15697.383} C_VEL
LIN {X 0,Y 312.492,Z 561.559,A -85,B 0,C 180,E1 -15700.709,E2 -15700.709} C_VEL
LIN {X 0,Y 312.454,Z 561.562,A -85,B 0,C 180,E1 -15704.21,E2 -15704.21} C_VEL
LIN {X 0,Y 312.486,Z 561.537,A -85,B 0,C 180,E1 -15707.919,E2 -15707.919} C_VEL
LIN {X 0,Y 312.499,Z 561.543,A -85,B 0,C 180,E1 -15711.834,E2 -15711.834} C_VEL
LIN {X 0,Y 312.518,Z 561.592,A -85,B 0,C 180,E1 -15711.915,E2 -15711.915} C_VEL
LIN {X 0,Y 316.44,Z 574.35,A -85,B 0,C 180,E1 -15714.935,E2 -15714.935} C_VEL
LIN {X 0,Y 320.12,Z 588.973,A -85,B 0,C 180,E1 -15718.203,E2 -15718.203} C_VEL
LIN {X 0,Y 322.062,Z 598.519,A -85,B 0,C 180,E1 -15720.207,E2 -15720.207} C_VEL
LIN {X 0,Y 320.538,Z 616.149,A -85,B 0,C 180,E1 -15723.289,E2 -15723.289} C_VEL
LIN {X 0,Y 319.977,Z 624.655,A -85,B 0,C 180,E1 -15724.702,E2 -15724.702} C_VEL
LIN {X 0,Y 324.555,Z 653.175,A -85,B 0,C 180,E1 -15725.771,E2 -15725.771} C_VEL
LIN {X 0,Y 323.078,Z 721.561,A -85,B 0,C 180,E1 -15727.286,E2 -15727.286} C_VEL
LIN {X 0,Y 322.631,Z 738.69,A -85,B 0,C 180,E1 -15727.717,E2 -15727.717} C_VEL
LIN {X 0,Y 321.804,Z 751.758,A -85,B 0,C 180,E1 -15728.29,E2 -15728.29} C_VEL
LIN {X 0,Y 320.807,Z 763.8,A -85,B 0,C 180,E1 -15729.061,E2 -15729.061} C_VEL
LIN {X 0,Y 319.682,Z 775.504,A -85,B 0,C 180,E1 -15730.076,E2 -15730.076} C_VEL
LIN {X 0,Y 318.403,Z 785.429,A -85,B 0,C 180,E1 -15731.166,E2 -15731.166} C_VEL
LIN {X 0,Y 317.08,Z 796.231,A -85,B 0,C 180,E1 -15732.667,E2 -15732.667} C_VEL
LIN {X 0,Y 315.725,Z 805.062,A -85,B 0,C 180,E1 -15734.175,E2 -15734.175} C_VEL
LIN {X 0,Y 314.256,Z 814.033,A -85,B 0,C 180,E1 -15736.088,E2 -15736.088} C_VEL
LIN {X 0,Y 313.132,Z 821.237,A -85,B 0,C 180,E1 -15738.017,E2 -15738.017} C_VEL
LIN {X 0,Y 312.102,Z 827.849,A -85,B 0,C 180,E1 -15740.276,E2 -15740.276} C_VEL
LIN {X 0,Y 311.534,Z 832.184,A -85,B 0,C 180,E1 -15742.22,E2 -15742.22} C_VEL
LIN {X 0,Y 311.264,Z 834.464,A -85,B 0,C 180,E1 -15743.517,E2 -15743.517} C_VEL
LIN {X 0,Y 311.058,Z 836.323,A -85,B 0,C 180,E1 -15744.814,E2 -15744.814} C_VEL
LIN {X 0,Y 310.915,Z 837.743,A -85,B 0,C 180,E1 -15746.111,E2 -15746.111} C_VEL
LIN {X 0,Y 310.696,Z 839.354,A -85,B 0,C 180,E1 -15748.703,E2 -15748.703} C_VEL
LIN {X 0,Y 310.696,Z 839.587,A -85,B 0,C 180,E1 -15749.999,E2 -15749.999} C_VEL
LIN {X 0,Y 310.695,Z 839.394,A -85,B 0,C 180,E1 -15751.295,E2 -15751.295} C_VEL
LIN {X 0,Y 310.909,Z 837.838,A -85,B 0,C 180,E1 -15753.887,E2 -15753.887} C_VEL
LIN {X 0,Y 311.055,Z 836.47,A -85,B 0,C 180,E1 -15755.184,E2 -15755.184} C_VEL
LIN {X 0,Y 311.347,Z 833.706,A -85,B 0,C 180,E1 -15757.065,E2 -15757.065} C_VEL
LIN {X 0,Y 311.859,Z 829.687,A -85,B 0,C 180,E1 -15759.075,E2 -15759.075} C_VEL
LIN {X 0,Y 312.616,Z 824.625,A -85,B 0,C 180,E1 -15761.015,E2 -15761.015} C_VEL
LIN {X 0,Y 313.599,Z 818.242,A -85,B 0,C 180,E1 -15762.949,E2 -15762.949} C_VEL
LIN {X 0,Y 314.912,Z 810.296,A -85,B 0,C 180,E1 -15764.87,E2 -15764.87} C_VEL
LIN {X 0,Y 316.26,Z 802.166,A -85,B 0,C 180,E1 -15766.458,E2 -15766.458} C_VEL
LIN {X 0,Y 317.599,Z 792.18,A -85,B 0,C 180,E1 -15768.046,E2 -15768.046} C_VEL
LIN {X 0,Y 319.02,Z 780.953,A -85,B 0,C 180,E1 -15769.462,E2 -15769.462} C_VEL
LIN {X 0,Y 320.311,Z 769.914,A -85,B 0,C 180,E1 -15770.551,E2 -15770.551} C_VEL
LIN {X 0,Y 321.508,Z 757.434,A -85,B 0,C 180,E1 -15771.477,E2 -15771.477} C_VEL
LIN {X 0,Y 322.267,Z 745.219,A -85,B 0,C 180,E1 -15772.138,E2 -15772.138} C_VEL
LIN {X 0,Y 322.825,Z 733.083,A -85,B 0,C 180,E1 -15772.562,E2 -15772.562} C_VEL
LIN {X 0,Y 324.577,Z 656.183,A -85,B 0,C 180,E1 -15774.266,E2 -15774.266} C_VEL
LIN {X 0,Y 320.544,Z 632.407,A -85,B 0,C 180,E1 -15775.17,E2 -15775.17} C_VEL
LIN {X 0,Y 319.182,Z 625.382,A -85,B 0,C 180,E1 -15775.475,E2 -15775.475} C_VEL
LIN {X 0,Y 320.499,Z 608.354,A -85,B 0,C 180,E1 -15778.701,E2 -15778.701} C_VEL
LIN {X 0,Y 321.419,Z 597.993,A -85,B 0,C 180,E1 -15780.774,E2 -15780.774} C_VEL
LIN {X 0,Y 319.633,Z 588.278,A -85,B 0,C 180,E1 -15783.033,E2 -15783.033} C_VEL
LIN {X 0,Y 318.176,Z 585.113,A -85,B 0,C 180,E1 -15783.884,E2 -15783.884} C_VEL
LIN {X 0,Y 310.889,Z 577.153,A -85,B 0,C 180,E1 -15786.491,E2 -15786.491} C_VEL
LIN {X 0,Y 309.064,Z 574.199,A -85,B 0,C 180,E1 -15787.388,E2 -15787.388} C_VEL
LIN {X 0,Y 308.68,Z 573.104,A -85,B 0,C 180,E1 -15787.688,E2 -15787.688} C_VEL
LIN {X 0,Y 305.451,Z 562.432,A -85,B 0,C 180,E1 -15790.598,E2 -15790.598} C_VEL
LIN {X 0,Y 305.478,Z 562.419,A -85,B 0,C 180,E1 -15794.643,E2 -15794.643} C_VEL
LIN {X 0,Y 313.793,Z 585.774,A -85,B 0,C 180,E1 -15795.838,E2 -15795.838} C_VEL
LIN {X 0,Y 312.567,Z 638.44,A -85,B 0,C 180,E1 -15797.323,E2 -15797.323} C_VEL
LIN {X 0,Y 312.411,Z 653.099,A -85,B 0,C 180,E1 -15797.912,E2 -15797.912} C_VEL
LIN {X 0,Y 311.969,Z 665.767,A -85,B 0,C 180,E1 -15798.673,E2 -15798.673} C_VEL
LIN {X 0,Y 311.256,Z 678.862,A -85,B 0,C 180,E1 -15799.742,E2 -15799.742} C_VEL
LIN {X 0,Y 310.576,Z 689.841,A -85,B 0,C 180,E1 -15800.892,E2 -15800.892} C_VEL
LIN {X 0,Y 309.754,Z 700.105,A -85,B 0,C 180,E1 -15802.222,E2 -15802.222} C_VEL
LIN {X 0,Y 308.844,Z 710.756,A -85,B 0,C 180,E1 -15803.928,E2 -15803.928} C_VEL
LIN {X 0,Y 308.031,Z 719.384,A -85,B 0,C 180,E1 -15805.619,E2 -15805.619} C_VEL
LIN {X 0,Y 307.372,Z 726.652,A -85,B 0,C 180,E1 -15807.357,E2 -15807.357} C_VEL
LIN {X 0,Y 306.703,Z 733.409,A -85,B 0,C 180,E1 -15809.346,E2 -15809.346} C_VEL
LIN {X 0,Y 306.344,Z 738.464,A -85,B 0,C 180,E1 -15811.199,E2 -15811.199} C_VEL
LIN {X 0,Y 305.952,Z 743.53,A -85,B 0,C 180,E1 -15813.615,E2 -15813.615} C_VEL
LIN {X 0,Y 305.81,Z 746.438,A -85,B 0,C 180,E1 -15815.564,E2 -15815.564} C_VEL
LIN {X 0,Y 305.855,Z 747.959,A -85,B 0,C 180,E1 -15817.006,E2 -15817.006} C_VEL
LIN {X 0,Y 305.945,Z 748.976,A -85,B 0,C 180,E1 -15818.436,E2 -15818.436} C_VEL
LIN {X 0,Y 306.23,Z 749.556,A -85,B 0,C 180,E1 -15820.207,E2 -15820.207} C_VEL
LIN {X 0,Y 306.835,Z 749.114,A -85,B 0,C 180,E1 -15822.677,E2 -15822.677} C_VEL
LIN {X 0,Y 307.337,Z 748.195,A -85,B 0,C 180,E1 -15824.073,E2 -15824.073} C_VEL
LIN {X 0,Y 307.902,Z 746.783,A -85,B 0,C 180,E1 -15825.458,E2 -15825.458} C_VEL
LIN {X 0,Y 308.552,Z 744.919,A -85,B 0,C 180,E1 -15826.834,E2 -15826.834} C_VEL
LIN {X 0,Y 309.703,Z 741.114,A -85,B 0,C 180,E1 -15828.879,E2 -15828.879} C_VEL
LIN {X 0,Y 311.37,Z 735.001,A -85,B 0,C 180,E1 -15831.269,E2 -15831.269} C_VEL
LIN {X 0,Y 312.949,Z 728.445,A -85,B 0,C 180,E1 -15833.229,E2 -15833.229} C_VEL
LIN {X 0,Y 314.773,Z 719.986,A -85,B 0,C 180,E1 -15835.197,E2 -15835.197} C_VEL
LIN {X 0,Y 316.404,Z 711.313,A -85,B 0,C 180,E1 -15836.817,E2 -15836.817} C_VEL
LIN {X 0,Y 318.006,Z 701.307,A -85,B 0,C 180,E1 -15838.326,E2 -15838.326} C_VEL
LIN {X 0,Y 319.604,Z 689.953,A -85,B 0,C 180,E1 -15839.685,E2 -15839.685} C_VEL
LIN {X 0,Y 320.85,Z 678.274,A -85,B 0,C 180,E1 -15840.784,E2 -15840.784} C_VEL
LIN {X 0,Y 321.801,Z 665.074,A -85,B 0,C 180,E1 -15841.721,E2 -15841.721} C_VEL
LIN {X 0,Y 322.274,Z 652.98,A -85,B 0,C 180,E1 -15842.343,E2 -15842.343} C_VEL
LIN {X 0,Y 323.059,Z 626.113,A -85,B 0,C 180,E1 -15843.251,E2 -15843.251} C_VEL
LIN {X 0,Y 324.629,Z 595.312,A -85,B 0,C 180,E1 -15844.221,E2 -15844.221} C_VEL
LIN {X 0,Y 319.253,Z 585.034,A -85,B 0,C 180,E1 -15845.414,E2 -15845.414} C_VEL
LIN {X 0,Y 310.83,Z 570.903,A -85,B 0,C 180,E1 -15847.418,E2 -15847.418} C_VEL
LIN {X 0,Y 308.854,Z 567.601,A -85,B 0,C 180,E1 -15847.941,E2 -15847.941} C_VEL
LIN {X 0,Y 306.517,Z 564.758,A -85,B 0,C 180,E1 -15848.524,E2 -15848.524} C_VEL
LIN {X 0,Y 305.775,Z 562.399,A -85,B 0,C 180,E1 -15848.803,E2 -15848.803} C_VEL
LIN {X 0,Y 305.58,Z 562.415,A -85,B 0,C 180,E1 -15853.296,E2 -15853.296} C_VEL
LIN {X 0,Y 305.584,Z 562.411,A -85,B 0,C 180,E1 -15856.021,E2 -15856.021} C_VEL
LIN {X 0,Y 305.568,Z 562.421,A -85,B 0,C 180,E1 -15859.446,E2 -15859.446} C_VEL
LIN {X 0,Y 305.481,Z 562.432,A -85,B 0,C 180,E1 -15863.042,E2 -15863.042} C_VEL
LIN {X 0,Y 305.539,Z 562.424,A -85,B 0,C 180,E1 -15866.228,E2 -15866.228} C_VEL
LIN {X 0,Y 305.488,Z 562.431,A -85,B 0,C 180,E1 -15869.051,E2 -15869.051} C_VEL
LIN {X 0,Y 305.457,Z 562.436,A -85,B 0,C 180,E1 -15873.518,E2 -15873.518} C_VEL
LIN {X 0,Y 305.49,Z 562.429,A -85,B 0,C 180,E1 -15876.737,E2 -15876.737} C_VEL
LIN {X 0,Y 305.489,Z 562.428,A -85,B 0,C 180,E1 -15880.61,E2 -15880.61} C_VEL
LIN {X 0,Y 305.557,Z 562.476,A -85,B 0,C 180,E1 -15884.329,E2 -15884.329} C_VEL
LIN {X 0,Y 307.717,Z 569.29,A -85,B 0,C 180,E1 -15887.613,E2 -15887.613} C_VEL
LIN {X 0,Y 309.988,Z 576.522,A -85,B 0,C 180,E1 -15890.596,E2 -15890.596} C_VEL
LIN {X 0,Y 312.583,Z 586.351,A -85,B 0,C 180,E1 -15894.038,E2 -15894.038} C_VEL
LIN {X 0,Y 314.472,Z 595.346,A -85,B 0,C 180,E1 -15896.803,E2 -15896.803} C_VEL
LIN {X 0,Y 315.104,Z 599.368,A -85,B 0,C 180,E1 -15897.946,E2 -15897.946} C_VEL
LIN {X 0,Y 314.41,Z 604.035,A -85,B 0,C 180,E1 -15899.063,E2 -15899.063} C_VEL
LIN {X 0,Y 313.422,Z 609.071,A -85,B 0,C 180,E1 -15900.212,E2 -15900.212} C_VEL
LIN {X 0,Y 316.831,Z 628.689,A -85,B 0,C 180,E1 -15901.539,E2 -15901.539} C_VEL
LIN {X 0,Y 319.257,Z 646.986,A -85,B 0,C 180,E1 -15902.583,E2 -15902.583} C_VEL
LIN {X 0,Y 320.943,Z 667.63,A -85,B 0,C 180,E1 -15903.571,E2 -15903.571} C_VEL
LIN {X 0,Y 321.376,Z 682.331,A -85,B 0,C 180,E1 -15904.164,E2 -15904.164} C_VEL
LIN {X 0,Y 319.16,Z 725.879,A -85,B 0,C 180,E1 -15905.486,E2 -15905.486} C_VEL
LIN {X 0,Y 317.84,Z 739.41,A -85,B 0,C 180,E1 -15906.115,E2 -15906.115} C_VEL
LIN {X 0,Y 316.139,Z 751.967,A -85,B 0,C 180,E1 -15906.934,E2 -15906.934} C_VEL
LIN {X 0,Y 315.066,Z 758.82,A -85,B 0,C 180,E1 -15907.458,E2 -15907.458} C_VEL
LIN {X 0,Y 314.153,Z 771.505,A -85,B 0,C 180,E1 -15908.081,E2 -15908.081} C_VEL
LIN {X 0,Y 312.951,Z 783.774,A -85,B 0,C 180,E1 -15908.943,E2 -15908.943} C_VEL
LIN {X 0,Y 311.597,Z 795.584,A -85,B 0,C 180,E1 -15910.055,E2 -15910.055} C_VEL
LIN {X 0,Y 309.993,Z 807.279,A -85,B 0,C 180,E1 -15911.496,E2 -15911.496} C_VEL
LIN {X 0,Y 308.551,Z 817.383,A -85,B 0,C 180,E1 -15913.068,E2 -15913.068} C_VEL
LIN {X 0,Y 307.227,Z 826.049,A -85,B 0,C 180,E1 -15914.749,E2 -15914.749} C_VEL
LIN {X 0,Y 305.929,Z 834.225,A -85,B 0,C 180,E1 -15916.72,E2 -15916.72} C_VEL
LIN {X 0,Y 304.983,Z 840.796,A -85,B 0,C 180,E1 -15918.706,E2 -15918.706} C_VEL
LIN {X 0,Y 304.326,Z 846.017,A -85,B 0,C 180,E1 -15920.698,E2 -15920.698} C_VEL
LIN {X 0,Y 303.932,Z 850.055,A -85,B 0,C 180,E1 -15922.695,E2 -15922.695} C_VEL
LIN {X 0,Y 303.721,Z 853.029,A -85,B 0,C 180,E1 -15924.69,E2 -15924.69} C_VEL
LIN {X 0,Y 303.72,Z 854.458,A -85,B 0,C 180,E1 -15926.021,E2 -15926.021} C_VEL
LIN {X 0,Y 303.69,Z 855.465,A -85,B 0,C 180,E1 -15927.348,E2 -15927.348} C_VEL
LIN {X 0,Y 303.675,Z 856.079,A -85,B 0,C 180,E1 -15928.675,E2 -15928.675} C_VEL
LIN {X 0,Y 303.727,Z 856.298,A -85,B 0,C 180,E1 -15930.001,E2 -15930.001} C_VEL
LIN {X 0,Y 303.684,Z 855.451,A -85,B 0,C 180,E1 -15932.654,E2 -15932.654} C_VEL
LIN {X 0,Y 303.712,Z 854.439,A -85,B 0,C 180,E1 -15933.982,E2 -15933.982} C_VEL
LIN {X 0,Y 303.774,Z 852.307,A -85,B 0,C 180,E1 -15935.826,E2 -15935.826} C_VEL
LIN {X 0,Y 304.043,Z 848.774,A -85,B 0,C 180,E1 -15937.973,E2 -15937.973} C_VEL
LIN {X 0,Y 304.487,Z 844.351,A -85,B 0,C 180,E1 -15939.97,E2 -15939.97} C_VEL
LIN {X 0,Y 305.178,Z 838.709,A -85,B 0,C 180,E1 -15941.963,E2 -15941.963} C_VEL
LIN {X 0,Y 306.307,Z 831.614,A -85,B 0,C 180,E1 -15943.941,E2 -15943.941} C_VEL
LIN {X 0,Y 307.697,Z 822.767,A -85,B 0,C 180,E1 -15945.909,E2 -15945.909} C_VEL
LIN {X 0,Y 308.982,Z 813.666,A -85,B 0,C 180,E1 -15947.541,E2 -15947.541} C_VEL
LIN {X 0,Y 310.447,Z 803.524,A -85,B 0,C 180,E1 -15948.992,E2 -15948.992} C_VEL
LIN {X 0,Y 311.952,Z 792.267,A -85,B 0,C 180,E1 -15950.267,E2 -15950.267} C_VEL
LIN {X 0,Y 313.25,Z 780.562,A -85,B 0,C 180,E1 -15951.296,E2 -15951.296} C_VEL
LIN {X 0,Y 314.437,Z 767.633,A -85,B 0,C 180,E1 -15952.116,E2 -15952.116} C_VEL
LIN {X 0,Y 315.289,Z 754.929,A -85,B 0,C 180,E1 -15952.658,E2 -15952.658} C_VEL
LIN {X 0,Y 315.968,Z 731.915,A -85,B 0,C 180,E1 -15953.211,E2 -15953.211} C_VEL
LIN {X 0,Y 316.97,Z 680.292,A -85,B 0,C 180,E1 -15954.379,E2 -15954.379} C_VEL
LIN {X 0,Y 313.806,Z 650.685,A -85,B 0,C 180,E1 -15955.369,E2 -15955.369} C_VEL
LIN {X 0,Y 311.706,Z 635.384,A -85,B 0,C 180,E1 -15955.945,E2 -15955.945} C_VEL
LIN {X 0,Y 310.356,Z 614.66,A -85,B 0,C 180,E1 -15957.637,E2 -15957.637} C_VEL
LIN {X 0,Y 309.71,Z 606.373,A -85,B 0,C 180,E1 -15958.333,E2 -15958.333} C_VEL
LIN {X 0,Y 311.591,Z 592.239,A -85,B 0,C 180,E1 -15961.629,E2 -15961.629} C_VEL
LIN {X 0,Y 311.307,Z 589.019,A -85,B 0,C 180,E1 -15962.424,E2 -15962.424} C_VEL
LIN {X 0,Y 308.363,Z 575.319,A -85,B 0,C 180,E1 -15965.998,E2 -15965.998} C_VEL
LIN {X 0,Y 305.49,Z 562.433,A -85,B 0,C 180,E1 -15969.531,E2 -15969.531} C_VEL
LIN {X 0,Y 305.444,Z 562.426,A -85,B 0,C 180,E1 -15973.652,E2 -15973.652} C_VEL
LIN {X 0,Y 305.462,Z 562.427,A -85,B 0,C 180,E1 -15977.414,E2 -15977.414} C_VEL
LIN {X 0,Y 305.469,Z 562.431,A -85,B 0,C 180,E1 -15981.596,E2 -15981.596} C_VEL
LIN {X 0,Y 305.464,Z 562.428,A -85,B 0,C 180,E1 -15984.887,E2 -15984.887} C_VEL
LIN {X 0,Y 305.453,Z 562.42,A -85,B 0,C 180,E1 -15988.355,E2 -15988.355} C_VEL
LIN {X 0,Y 305.522,Z 562.424,A -85,B 0,C 180,E1 -15991.114,E2 -15991.114} C_VEL
LIN {X 0,Y 305.573,Z 562.409,A -85,B 0,C 180,E1 -15994.088,E2 -15994.088} C_VEL
LIN {X 0,Y 305.483,Z 562.431,A -85,B 0,C 180,E1 -15998.402,E2 -15998.402} C_VEL
LIN {X 0,Y 305.591,Z 562.399,A -85,B 0,C 180,E1 -16001.218,E2 -16001.218} C_VEL
LIN {X 0,Y 305.65,Z 562.411,A -85,B 0,C 180,E1 -16005.349,E2 -16005.349} C_VEL
LIN {X 0,Y 305.637,Z 562.388,A -85,B 0,C 180,E1 -16009.4,E2 -16009.4} C_VEL
LIN {X 0,Y 305.799,Z 562.389,A -85,B 0,C 180,E1 -16012.074,E2 -16012.074} C_VEL
LIN {X 0,Y 305.688,Z 562.403,A -85,B 0,C 180,E1 -16014.723,E2 -16014.723} C_VEL
LIN {X 0,Y 305.956,Z 562.357,A -85,B 0,C 180,E1 -16018.684,E2 -16018.684} C_VEL
LIN {X 0,Y 305.958,Z 562.374,A -85,B 0,C 180,E1 -16021.316,E2 -16021.316} C_VEL
LIN {X 0,Y 305.848,Z 562.374,A -85,B 0,C 180,E1 -16026.598,E2 -16026.598} C_VEL
LIN {X 0,Y 305.738,Z 562.401,A -85,B 0,C 180,E1 -16029.26,E2 -16029.26} C_VEL
LIN {X 0,Y 305.59,Z 562.399,A -85,B 0,C 180,E1 -16033.296,E2 -16033.296} C_VEL
LIN {X 0,Y 305.596,Z 562.42,A -85,B 0,C 180,E1 -16036.02,E2 -16036.02} C_VEL
LIN {X 0,Y 305.578,Z 562.399,A -85,B 0,C 180,E1 -16039.445,E2 -16039.445} C_VEL
LIN {X 0,Y 305.493,Z 562.43,A -85,B 0,C 180,E1 -16043.041,E2 -16043.041} C_VEL
LIN {X 0,Y 305.528,Z 562.413,A -85,B 0,C 180,E1 -16046.219,E2 -16046.219} C_VEL
LIN {X 0,Y 305.49,Z 562.43,A -85,B 0,C 180,E1 -16049.047,E2 -16049.047} C_VEL
LIN {X 0,Y 305.445,Z 562.43,A -85,B 0,C 180,E1 -16051.952,E2 -16051.952} C_VEL
LIN {X 0,Y 305.464,Z 562.426,A -85,B 0,C 180,E1 -16055.113,E2 -16055.113} C_VEL
LIN {X 0,Y 305.469,Z 562.434,A -85,B 0,C 180,E1 -16058.533,E2 -16058.533} C_VEL
LIN {X 0,Y 305.457,Z 562.431,A -85,B 0,C 180,E1 -16062.586,E2 -16062.586} C_VEL
LIN {X 0,Y 305.428,Z 562.421,A -85,B 0,C 180,E1 -16066.345,E2 -16066.345} C_VEL
LIN {X 0,Y 305.461,Z 562.439,A -85,B 0,C 180,E1 -16069.892,E2 -16069.892} C_VEL
LIN {X 0,Y 305.488,Z 562.6,A -85,B 0,C 180,E1 -16071.201,E2 -16071.201} C_VEL
LIN {X 0,Y 309.47,Z 575.421,A -85,B 0,C 180,E1 -16074.339,E2 -16074.339} C_VEL
LIN {X 0,Y 312.992,Z 588.741,A -85,B 0,C 180,E1 -16077.39,E2 -16077.39} C_VEL
LIN {X 0,Y 315.431,Z 600.497,A -85,B 0,C 180,E1 -16079.913,E2 -16079.913} C_VEL
LIN {X 0,Y 313.832,Z 618.209,A -85,B 0,C 180,E1 -16083.032,E2 -16083.032} C_VEL
LIN {X 0,Y 313.36,Z 624.753,A -85,B 0,C 180,E1 -16084.126,E2 -16084.126} C_VEL
LIN {X 0,Y 317.673,Z 650.907,A -85,B 0,C 180,E1 -16085.153,E2 -16085.153} C_VEL
LIN {X 0,Y 318.145,Z 656.11,A -85,B 0,C 180,E1 -16085.32,E2 -16085.32} C_VEL
LIN {X 0,Y 316.178,Z 736.294,A -85,B 0,C 180,E1 -16087.151,E2 -16087.151} C_VEL
LIN {X 0,Y 315.492,Z 749.022,A -85,B 0,C 180,E1 -16087.66,E2 -16087.66} C_VEL
LIN {X 0,Y 314.456,Z 761.83,A -85,B 0,C 180,E1 -16088.445,E2 -16088.445} C_VEL
LIN {X 0,Y 313.19,Z 774.062,A -85,B 0,C 180,E1 -16089.474,E2 -16089.474} C_VEL
LIN {X 0,Y 311.854,Z 784.342,A -85,B 0,C 180,E1 -16090.584,E2 -16090.584} C_VEL
LIN {X 0,Y 310.635,Z 793.698,A -85,B 0,C 180,E1 -16091.849,E2 -16091.849} C_VEL
LIN {X 0,Y 309.214,Z 803.517,A -85,B 0,C 180,E1 -16093.494,E2 -16093.494} C_VEL
LIN {X 0,Y 307.6,Z 812.89,A -85,B 0,C 180,E1 -16095.443,E2 -16095.443} C_VEL
LIN {X 0,Y 306.362,Z 820.339,A -85,B 0,C 180,E1 -16097.411,E2 -16097.411} C_VEL
LIN {X 0,Y 305.376,Z 826.32,A -85,B 0,C 180,E1 -16099.39,E2 -16099.39} C_VEL
LIN {X 0,Y 304.669,Z 831.046,A -85,B 0,C 180,E1 -16101.376,E2 -16101.376} C_VEL
LIN {X 0,Y 304.193,Z 834.784,A -85,B 0,C 180,E1 -16103.447,E2 -16103.447} C_VEL
LIN {X 0,Y 303.977,Z 836.517,A -85,B 0,C 180,E1 -16104.693,E2 -16104.693} C_VEL
